// TIA Portal V19 program export: 4 tag tables, 24 data types, 99 data blocks, 53 code blocks (in call order from the OBs), 0 instance data blocks

VAR_GLOBAL   // PLC tag table "Default tag table"
   Tag_111 AT %MW1 : Int;
   di_1 AT %I0.0 : Bool;
   di_2 AT %I0.1 : Bool;
   ai_raw_01 AT %IW272 : Int;
   ai_raw_02 AT %IW274 : Int;
   ai_raw_03 AT %IW276 : Int;
   ai_raw_04 AT %IW278 : Int;
END_VAR
VAR_GLOBAL CONSTANT   // user constants
   C_HW_MAX : Int := 27648;
   C_HW_MIN : Int := 0;
   C_DIAG_OVER : Real := 1.1759;
   C_DIAG_UNDER : Real := -0.1759;
END_VAR

VAR_GLOBAL   // PLC tag table "Tag table_1"
   r1 AT %M20.0 : Bool;
   tr1 AT %M20.1 : Bool;
   r2 AT %M20.2 : Bool;
   tr2 AT %M20.3 : Bool;
   r3 AT %M20.4 : Bool;
   tr3 AT %M20.5 : Bool;
   r4 AT %M20.6 : Bool;
   tr4 AT %M20.7 : Bool;
   r5 AT %M21.0 : Bool;
   tr5 AT %M21.1 : Bool;
   r6 AT %M21.2 : Bool;
   tr6 AT %M21.3 : Bool;
   r7 AT %M21.4 : Bool;
   tr7 AT %M21.5 : Bool;
   r8 AT %M21.6 : Bool;
   tr8 AT %M21.7 : Bool;
   r9 AT %M22.0 : Bool;
   tr9 AT %M22.1 : Bool;
   r10 AT %M22.2 : Bool;
   tr10 AT %M22.3 : Bool;
   r11 AT %M22.4 : Bool;
   tr11 AT %M22.5 : Bool;
   r12 AT %M22.6 : Bool;
   tr12 AT %M22.7 : Bool;
   r13 AT %M23.0 : Bool;
   tr13 AT %M23.1 : Bool;
   r14 AT %M23.2 : Bool;
   tr14 AT %M23.3 : Bool;
   r15 AT %M23.4 : Bool;
   tr15 AT %M23.5 : Bool;
END_VAR

VAR_GLOBAL   // PLC tag table "Tag table_2"
   Pol_sklad_sens AT %IW40 : Int;
   Pol_sens AT %IW42 : Int;
END_VAR

VAR_GLOBAL   // PLC tag table "Tag tanks"
END_VAR
VAR_GLOBAL CONSTANT   // user constants
   c_Count_TRN : Int := 3;
   c_Count_POL : Int := 10;
   c_Count_BUL : Int := 4;
   c_Count_MOL : Int := 12;
END_VAR

TYPE "UDT_AI_Alarm_Conf"
VERSION : 0.1
   STRUCT
      En_Alarm : Struct
         HiHi { S7_SetPoint := 'True'} : Bool;
         Hi { S7_SetPoint := 'True'} : Bool;
         Lo { S7_SetPoint := 'True'} : Bool;
         LoLo { S7_SetPoint := 'True'} : Bool;
         Latch_Enable { S7_SetPoint := 'True'} : Bool;   // 1 = Включена фиксация аварий (до нажатия Reset)
         Pad_Bit_5 { S7_SetPoint := 'True'} : Bool;   // Резерв
         Pad_Bit_6 { S7_SetPoint := 'True'} : Bool;   // Резерв
         Pad_Bit_7 { S7_SetPoint := 'True'} : Bool;   // Резерв
      END_STRUCT;
      HiHi { S7_SetPoint := 'True'} : Real;
      Hi { S7_SetPoint := 'True'} : Real;
      Lo { S7_SetPoint := 'True'} : Real;
      LoLo { S7_SetPoint := 'True'} : Real;
      Delay_HiHi { S7_SetPoint := 'True'} : Int;
      Delay_Hi { S7_SetPoint := 'True'} : Int;
      Delay_Lo { S7_SetPoint := 'True'} : Int;
      Delay_LoLo { S7_SetPoint := 'True'} : Int;
      Hysteresis { S7_SetPoint := 'True'} : Real;
   END_STRUCT;

END_TYPE

TYPE "UDT_AI_Conf"
VERSION : 0.1
   STRUCT
      Mode { S7_SetPoint := 'True'} : Word := 16#0010;   // ПО УМОЛЧАНИЮ: Взведен Bit 4 (Final Clamp)
      Scale_Min { S7_SetPoint := 'True'} : Real := 0.0;   // Мин. физической шкалы
      Scale_Max { S7_SetPoint := 'True'} : Real := 100.0;   // Макс. физической шкалы
      Calib_mA_Min { S7_SetPoint := 'True'} : Real := 4.0;   // Ток при Scale_Min
      Calib_mA_Max { S7_SetPoint := 'True'} : Real := 20.0;   // Ток при Scale_Max
      Cutoff { S7_SetPoint := 'True'} : Real := 0.02;   // Порог отсечения шума около нуля
      FilterTime_ms { S7_SetPoint := 'True'} : Int := 2000;   // Время фильтра PT1 в миллисекундах (0..32000) --- Границы железа ---
      HW_Min { S7_SetPoint := 'True'} : Int := "C_HW_MIN";   // Аппаратный минимум
      HW_Max { S7_SetPoint := 'True'} : Int := "C_HW_MAX";   // Аппаратный максимум
   END_STRUCT;

END_TYPE

TYPE "UDT_AI_Config"
VERSION : 0.1
   STRUCT
      Mode : Word := 16#0010;   // ПО УМОЛЧАНИЮ: Взведен Bit 4 (Final Clamp)
      Scale_Min : Real := 0.0;   // Мин. физической шкалы
      Scale_Max : Real := 100.0;   // Макс. физической шкалы
      Calib_mA_Min : Real := 4.0;   // Ток при Scale_Min
      Calib_mA_Max : Real := 20.0;   // Ток при Scale_Max
      Cutoff : Real := 0.02;   // Порог отсечения шума около нуля
      FilterTime_ms : Int := 2000;   // Время фильтра PT1 в миллисекундах (0..32000) --- Границы железа ---
      HW_Min : Int := "C_HW_MIN";   // Аппаратный минимум
      HW_Max : Int := "C_HW_MAX";   // Аппаратный максимум
   END_STRUCT;

END_TYPE

TYPE "UDT_AI_Out"
VERSION : 0.1
   STRUCT
      Raw : Int;   // Сырой код с модуля (PIW)
      Value_mA : Real;   // Расчетный ток (мА)
      Value_Unclamped : Real;   // Чистая физика (ДО клампа и ДО фильтра)
      Value_Scaled : Real;   // Физика ПОСЛЕ клампа (ограниченная шкалой)
      Value_Filtered : Real;   // Финальное сглаженное значение (для HMI и алармов)
      Status : Struct
         WireBreak : Bool;
         Underrange : Bool;
         Overrange : Bool;
         Overflow : Bool;
         Sim_Active : Bool;
         ConfigError : Bool;
         Pad_Bit_6 : Bool;   // Выравнивание
         Pad_Bit_7 : Bool;   // Выравнивание
         Pad_Byte : Byte;   // Выравнивание структуры до 1 Word
      END_STRUCT;
   END_STRUCT;

END_TYPE

TYPE "UDT_AI_Status"
VERSION : 0.1
// -----------------------------------------------------------------------------
// 2. АВТОНОМНЫЙ СТАТУС (2 БАЙТА / 1 WORD)
// -----------------------------------------------------------------------------
   STRUCT
      WireBreak : Bool;   // +0.0 | Wire break (< -4864)
      Underrange : Bool;   // +0.1 | Signal < 0 mA, but alive
      Overrange : Bool;   // +0.2 | Signal > 20 mA
      Overflow : Bool;   // +0.3 | Short circuit (> 22.8 mA)
      Sim_Active : Bool;   // +0.4 | Simulation mode ON
      ConfigError : Bool;   // +0.5 | Bad settings in UDT_Config
      Pad_Bit_6 : Bool;   // +0.6
      Pad_Bit_7 : Bool;   // +0.7
      Pad_Byte : Byte;   // +1.0 | Alignment for S7-300
   END_STRUCT;

END_TYPE

TYPE "UDT_Alarm_Config"
VERSION : 1.0
   STRUCT
      En_Alarm : Struct
         HiHi         : Bool;
         Hi           : Bool;
         Lo           : Bool;
         LoLo         : Bool;
         Latch_Enable : Bool;  // 1 = Включена фиксация аварий (до нажатия Reset)
         Pad_Bit_5    : Bool;  // Резерв
         Pad_Bit_6    : Bool;  // Резерв
         Pad_Bit_7    : Bool;  // Резерв
      END_STRUCT;
      HiHi       : Real;
      Hi         : Real;
      Lo         : Real;
      LoLo       : Real;
      Delay_HiHi : Int;
      Delay_Hi   : Int;
      Delay_Lo   : Int;
      Delay_LoLo : Int;
      Hysteresis : Real;
   END_STRUCT;
END_TYPE

TYPE "UDT_Alarm_Out"
VERSION : 2.0
   STRUCT
      // --- Байт 0 (Аварии) ---
      HiHi         : Bool;
      Hi           : Bool;
      Lo           : Bool;
      LoLo         : Bool;
      Pad_Bit_4    : Bool; // Резерв
      Pad_Bit_5    : Bool; // Резерв
      Pad_Bit_6    : Bool; // Резерв
      Pad_Bit_7    : Bool; // Резерв
      
      // --- Байт 1 (Статусы для HMI) ---
      En_HiHi         : Bool;
      En_Hi           : Bool;
      En_Lo           : Bool;
      En_LoLo         : Bool;
      En_Latch_Enable : Bool; // Статус фиксации
      En_Pad_Bit_5    : Bool; // Резерв
      En_Pad_Bit_6    : Bool; // Резерв
      En_Pad_Bit_7    : Bool; // Резерв
   END_STRUCT;
END_TYPE

TYPE "UDT_DI_Alarm_Conf"
VERSION : 0.1
// =============================================================================
// СТРУКТУРЫ ДЛЯ ДИСКРЕТНОГО АЛАРМА (FB_DI_Alarm)
// =============================================================================
   STRUCT
      En_Alarm : Bool;   // 1 = Разрешение контроля аварии
      Invert : Bool;   // 0 = NO (TRUE = Авария), 1 = NC (FALSE = Авария)
      Latch_Enable : Bool;   // 1 = Фиксация аварии (требует сброса кнопкой Reset)
      Pad_Bit_3 : Bool;   // Резерв
      Pad_Bit_4 : Bool;   // Резерв
      Pad_Bit_5 : Bool;   // Резерв
      Pad_Bit_6 : Bool;   // Резерв
      Pad_Bit_7 : Bool;   // Резерв
      Pad_Byte : Byte;   // Выравнивание
      Delay : Int;   // Задержка срабатывания (в СЕКУНДАХ)
   END_STRUCT;

END_TYPE

TYPE "UDT_DI_Conf"
VERSION : 0.1
   STRUCT
      Mode { S7_SetPoint := 'True'} : Int;   // Режим: 0=Прямой, 1=С фильтром (Прямой), 2=С фильтром (Инверсный)
      FilterTime { S7_SetPoint := 'True'} : Int;   // Время антидребезга (мс), макс. 32767 мс
   END_STRUCT;

END_TYPE

TYPE "UDT_DI_Out"
VERSION : 0.1
// =============================================================================
// СТРУКТУРЫ ДЛЯ ОБРАБОТКИ ДИСКРЕТНОГО ВХОДА (FB_DI)
// =============================================================================
   STRUCT
      Value : Bool;   // Обработанное состояние входа (после антидребезга)
      Pad_Bit_1 : Bool;   // Резерв
      Pad_Bit_2 : Bool;   // Резерв
      Pad_Bit_3 : Bool;   // Резерв
      Pad_Bit_4 : Bool;   // Резерв
      Pad_Bit_5 : Bool;   // Резерв
      Pad_Bit_6 : Bool;   // Резерв
      Pad_Bit_7 : Bool;   // Резерв
      Pad_Byte : Byte;   // Выравнивание до слова (Word) для SCADA
   END_STRUCT;

END_TYPE

TYPE "UDT_HMI_SmallTank"
TITLE = Данные малого танка для HMI
VERSION : 0.1
//Описание:
//        Плоская структура малого танка для обмена с панелью оператора.
//        Статусные слова развернуты побитово с жестким выравниванием 
//        до 16 бит (WORD) для прямого маппинга в библиотеку WinCC.
   STRUCT
      Level_m : Real;   // Текущий уровень
      Volume_m3 : Real;   // Рассчитанный объем
      Weight_t : Real;   // Рассчитанная масса в тоннах
      Percent_prc : Real;   // Уровень в процентах --- Развернутое слово Status_Alarms (Ровно 2 байта) ---
      Status_Alarms : Struct
         DI : Bool;   // ПЛК Бит 0.0 -> WinCC Бит 8
         HH : Bool;   // ПЛК Бит 0.1 -> WinCC Бит 9
         H : Bool;   // ПЛК Бит 0.2 -> WinCC Бит 10
         L : Bool;   // ПЛК Бит 0.3 -> WinCC Бит 11
         LL : Bool;   // ПЛК Бит 0.4 -> WinCC Бит 12
         Pad_0_5 : Bool;   // Выравнивание
         Pad_0_6 : Bool;   // Выравнивание
         Pad_0_7 : Bool;   // Выравнивание
         Pad_Byte : Byte;   // Резервный младший байт (WinCC Биты 0..7) --- Развернутое слово Status_AI (Ровно 2 байта) ---
      END_STRUCT;
      Status_AI : Struct
         WireBreak : Bool;   // ПЛК Бит 0.0 -> WinCC Бит 8
         Underrange : Bool;   // ПЛК Бит 0.1 -> WinCC Бит 9
         Overrange : Bool;   // ПЛК Бит 0.2 -> WinCC Бит 10
         Overflow : Bool;   // ПЛК Бит 0.3 -> WinCC Бит 11
         ConfigError : Bool;   // ПЛК Бит 0.4 -> WinCC Бит 12
         Pad_0_5 : Bool;   // Выравнивание
         Pad_0_6 : Bool;   // Выравнивание
         Pad_0_7 : Bool;   // Выравнивание
         Pad_Byte : Byte;   // Резервный младший байт (WinCC Биты 0..7) --- Развернутое слово Cmd_Word (Ровно 2 байта) ---
      END_STRUCT;
      Cmd : Struct
         Reset : Bool;   // ПЛК Бит 0.0 -> WinCC Бит 8 (Кнопка сброса)
         Pad_0_1 : Bool;   // Выравнивание
         Pad_0_2 : Bool;   // Выравнивание
         Pad_0_3 : Bool;   // Выравнивание
         Pad_0_4 : Bool;   // Выравнивание
         Pad_0_5 : Bool;   // Выравнивание
         Pad_0_6 : Bool;   // Выравнивание
         Pad_0_7 : Bool;   // Выравнивание
         Pad_Byte : Byte;   // Резервный младший байт (WinCC Биты 0..7)
      END_STRUCT;
      Spare_Real_1 : Real;   // Резерв для сохранения смещений
   END_STRUCT;

END_TYPE

TYPE "UDT_HMI_Whouse"
TITLE = Сводка склада для HMI
{ S7_Optimized_Access := 'FALSE' }
AUTHOR : S7A_Lib
FAMILY : HMI_Type
VERSION : 0.1
// ==============================================================================
// Описание: Агрегированные данные склада (тоталы, счетчики, глобальные 
//           статусы) для отображения на главном экране WinCC.
// ==============================================================================
    STRUCT
        Total_Volume_m3 : REAL;   // Суммарный объем продукта на складе
        Total_Weight_t : REAL;    // Суммарная масса (тонны)
        Total_Ullage_m3 : REAL;   // Доступное свободное место (м3)
        Tanks_In_Alarm : INT;     // Количество танков в состоянии аварии
        
        // --- Глобальные статусы склада (Ровно 2 байта) ---
        Status_Word : STRUCT 
            Comm_Error : BOOL;    // ПЛК Бит 0.0 -> WinCC Бит 8 (Ошибка связи с периферией)
            Global_Alarm : BOOL;  // ПЛК Бит 0.1 -> WinCC Бит 9 (Есть активные аварии)
            Pad_0_2 : BOOL;       // Выравнивание
            Pad_0_3 : BOOL;       // Выравнивание
            Pad_0_4 : BOOL;       // Выравнивание
            Pad_0_5 : BOOL;       // Выравнивание
            Pad_0_6 : BOOL;       // Выравнивание
            Pad_0_7 : BOOL;       // Выравнивание
            Pad_Byte : BYTE;      // Резервный младший байт (WinCC Биты 0..7)
        END_STRUCT;
        
        // --- Глобальные команды склада (Ровно 2 байта) ---
        Cmd_Word : STRUCT
            Reset_All : BOOL;     // ПЛК Бит 0.0 -> WinCC Бит 8 (Глобальный сброс аварий)
            Pad_0_1 : BOOL;       // Выравнивание
            Pad_0_2 : BOOL;       // Выравнивание
            Pad_0_3 : BOOL;       // Выравнивание
            Pad_0_4 : BOOL;       // Выравнивание
            Pad_0_5 : BOOL;       // Выравнивание
            Pad_0_6 : BOOL;       // Выравнивание
            Pad_0_7 : BOOL;       // Выравнивание
            Pad_Byte : BYTE;      // Резервный младший байт (WinCC Биты 0..7)
        END_STRUCT;
        
        Spare_Real_1 : REAL;      // Резерв для сохранения смещений
    END_STRUCT;
END_TYPE

TYPE "UDT_SIWA_CS"
VERSION : 0.0
   STRUCT
      i_DB_Lenght : Int := 222;
      i_MaxLifeBitCyc : Int := 500;
      i_SFC_ERR_C : Word;
      i_CMD_INPUT : Int;
      bo_CMD_TRIGGER : Bool;
      bo_CMD_IN_PROGRESS : Bool;
      bo_CMD_FINISHED_OK : Bool;
      bo_CMD_ERR : Bool;
      b_CMD_ERR_CODE : Byte;
      i_PRESET_TARE : Int;
      b_SELECT_PROC_VAL : Byte;
      b_SELECTED_PROC_VAL : Byte;
      i_PROCESS_VALUE : Int;
      b_INFO_REFRESH_COUNT : Byte;
      w_SCALE_STATUS : Word;
      b_OPR_ERR_MSG : Byte;
      bo_FB_ERR : Bool;
      b_FB_ERR_CODE : Byte;
      bo_START_UP_IN_PROGRESS : Bool;
      s_CMD1 : Struct
         i_CMD1_Code : Int;
         bo_CMD1_Trigger : Bool;
         bo_CMD1_InProgress : Bool;
         bo_CMD1_FinishedOk : Bool;
         bo_CMD1_FinishedError : Bool;
      END_STRUCT;
      s_CMD2 : Struct
         i_CMD2_Code : Int;
         bo_CMD2_Trigger : Bool;
         bo_CMD2_InProgress : Bool;
         bo_CMD2_FinishedOk : Bool;
         bo_CMD2_FinishedError : Bool;
      END_STRUCT;
      s_CMD3 : Struct
         i_CMD3_Code : Int;
         bo_CMD3_Trigger : Bool;
         bo_CMD3_InProgress : Bool;
         bo_CMD3_FinishedOk : Bool;
         bo_CMD3_FinishedError : Bool;
      END_STRUCT;
      w_DB_RES92 : Word;
      w_DB_RES93 : Word;
      w_DB_RES94 : Word;
      w_DB_RES95 : Word;
      w_DB_RES96 : Word;
      w_DB_RES97 : Word;
      w_INT_USE : Word;
      s_JUST_DAT : Struct
         w_CALIB_DIGITS0 : Word;
         w_CALIB_DIGITS1 : Word := W#16#EA60;
         w_CALIB_DIGITS2 : Word;
         i_CALIB_WEIGHT1 : Int := 2000;
         i_CALIB_WEIGHT2 : Int;
         b_SIGNAL_RANGE : Byte := B#16#2;
         b_FILT_TYPE : Byte;
         b_FILT_FREQ : Byte := B#16#4;
         b_FILT_DEPTH : Byte := B#16#F;
         s_SCALE_ID : String[10] := 'SIWAREX XX';
         i_MIN_WR : Int := 20;
         i_MAX_WR : Int := 2000;
         i_INCREMENT_WR : Int := 1;
         i_WEIGHT_ST_STILL : Int := 10;
         t_TIME_ST_STILL1 : Time := T#1S;
         b_DEC_POINT : Byte := B#16#2;
         b_ZERO_NEG_VALUE : Byte := B#16#1;
         b_ZERO_POS_VALUE : Byte := B#16#3;
         b_TARA_MAX : Byte := B#16#64;
         i_Reserve : Int;
         s_LEGAL_TRADE : String[4] := '----';
         s_WEGHT_UNIT : String[4] := 'kg  ';
      END_STRUCT;
      s_LIMIT_PARA : Struct
         i_LIMIT1_ON : Int := 400;
         i_LIMIT1_OFF : Int := 220;
         i_LIMIT2_ON : Int := 1000;
         i_LIMIT2_OFF : Int := 980;
         bo_LIMIT1_PARA : Bool;
         bo_LIMIT2_PARA : Bool;
         b_Reserve : Byte;
      END_STRUCT;
      s_MODUL_INFO_DATA : Struct
         s_MODUL_NAME : String[10];
         s_ORDER_NUM : String[20];
         w_VERSION_HW : Word;
         s_VERSION_FW : String[4];
         w_CRC_CHECK : Word;
      END_STRUCT;
      s_TARE_CONTROL : Struct
         i_TARE_VALUE : Int;
      END_STRUCT;
      s_INTERNAL_PROC_VAL : Struct
         w_CRC_CHECK : Word;
         b_Reserve : Byte;
         bo_PRESET_TARA : Bool;
         d_TARA_X_100 : DInt;
         d_ZERO_X_100 : DInt;
      END_STRUCT;
      s_PROCESS_VALUES : Struct
         w_CRC_CHECK : Word;
         bo_STA_WRI_PROT : Bool;
         bo_STA_WR_MIN : Bool;
         bo_STA_Reserve1 : Bool;
         bo_STA_Reserve2 : Bool;
         bo_STA_Reserve3 : Bool;
         bo_STA_Reserve4 : Bool;
         bo_STA_Reserve5 : Bool;
         bo_STA_ERROR_ON : Bool;
         bo_STA_LIMIT1_ON : Bool;
         bo_STA_LIMIT2_ON : Bool;
         bo_STA_TARED : Bool;
         bo_STA_TARED_BY_MANUAL : Bool;
         bo_STA_MAX_9E : Bool;
         bo_STA_025_D_ZERO : Bool;
         bo_STA_ST_STAND_SCALE_ON : Bool;
         bo_STA_SCALE_CALIBRATED : Bool;
         b_OPR_ERR_MSG : Byte;
         b_Reserve : Byte;
         i_GROSS_WEIGHT_PROC : Int;
         i_NET_WEIGHT_PROC : Int;
         i_TARE_WEIGHT_PROC : Int;
         i_GROSS_NET_VALUE : Int;
         d_GROSS_NET_VALUE_10X : DInt;
         i_TARE_VALUE : Int;
         i_ADC_DIGIT : Int;
         i_ADC_DIGIT_FILTER : Int;
         s_WEIGHT_ASCII : String[14];
         i_MILISEC : Int;
         b_SECONDS : Byte;
         b_MINUTE : Byte;
         i_HOURS : Int;
      END_STRUCT;
      i_DB_Lenght1 : Int := 222;
   END_STRUCT;

END_TYPE

TYPE "UDT_Siwarex_Core"
TITLE = Данные весового модуля Siwarex
VERSION : 0.2
//Описание:
//        Базовая структура для работы с весовыми модулями Siwarex.
//        Разделены операционные ошибки (модуля) и ошибки драйвера (FB).
    STRUCT
        Weight_Gross_kg : REAL;    // Брутто (полный вес)
        Weight_Net_kg : REAL;      // Нетто (чистый вес продукта)
        Weight_Tare_kg : REAL;     // Тара (вес пустой емкости)
        
        // --- Диагностика: Аппаратная ошибка модуля (из b_OPR_ERR_MSG) ---
        // 17 - Выход за максимальный предел взвешивания.
        // 19 - Перегруз АЦП (ADC overrange).
        // 20 - Недогруз АЦП (сигнал ушел далеко в минус).
        // 22 - Ошибка команды: весы не стабильны (жидкость плещется).
        // 31 - Обрыв провода тензодатчика (Wire break).
        Error_Op_Msg : INT;        
        
        // --- Диагностика: Ошибка драйвера ПЛК (из b_FB_ERR_CODE) ---
        // 1 - Watchdog тайм-аут (нет ответа от модуля на запрос данных).
        // 2 - Ошибка системной функции (SFC) RD_REC или WR_REC.
        // 3 - Некорректный номер команды в буфере или неверная длина DB.
        Error_FB_Code : INT;       
        
        // --- Статусы весов (Ровно 2 байта) ---
        Status : STRUCT
            Standstill : BOOL;     // ПЛК Бит 0.0 -> WinCC Бит 8 (Весы в покое)
            Limit_1 : BOOL;        // ПЛК Бит 0.1 -> WinCC Бит 9 (Предел 1)
            Limit_2 : BOOL;        // ПЛК Бит 0.2 -> WinCC Бит 10 (Предел 2)
            Fault_HW : BOOL;       // ПЛК Бит 0.3 -> WinCC Бит 11 (Аппаратная ошибка)
            Limit_Max : BOOL;      // ПЛК Бит 0.4 -> WinCC Бит 12 (Перегруз)
            Comm_Fault : BOOL;     // ПЛК Бит 0.5 -> WinCC Бит 13 (Watchdog: потеря связи)
            Fault_FB : BOOL;       // ПЛК Бит 0.6 -> WinCC Бит 14 (Ошибка драйвера)
            Pad_0_7 : BOOL;        // Выравнивание
            Pad_Byte : BYTE;       // Резервный младший байт (WinCC Биты 0..7)
        END_STRUCT;
        
        // --- Команды с HMI (Ровно 2 байта) ---
        Cmd : STRUCT
            Zero : BOOL;           // ПЛК Бит 0.0 -> WinCC Бит 8 (Установка нуля)
            Tare : BOOL;           // ПЛК Бит 0.1 -> WinCC Бит 9 (Тарирование)
            ResetError : BOOL;     // ПЛК Бит 0.2 -> WinCC Бит 10 (Сброс ошибки)
            Pad_0_3 : BOOL;        // Выравнивание
            Pad_0_4 : BOOL;        // Выравнивание
            Pad_0_5 : BOOL;        // Выравнивание
            Pad_0_6 : BOOL;        // Выравнивание
            Pad_0_7 : BOOL;        // Выравнивание
            Pad_Byte : BYTE;       // Резервный младший байт (WinCC Биты 0..7)
        END_STRUCT;
        
        Spare_Real_1 : REAL;       // Резерв
    END_STRUCT;
END_TYPE

TYPE "UDT_Sys_Info"
VERSION : 0.1
// ===============================================================
// Master Project: S7C_Master_AI_Test (S7-300 COMPLIANT)
// Platform: S7-300 / IM 151-8
// FIX: No FBs in Temp/Global DB. Using Multi-instance in Wrapper FB.
// Encoding: UTF-8 with BOM
// ===============================================================
// 1. DATA TYPES (UDTs)
   STRUCT
      FirstScan { ExternalVisible := 'False'} : Bool;
      CycleTime_ms_INT { ExternalVisible := 'False'} : Int;
      CycleTime_ms_REAL { ExternalVisible := 'False'} : Real;
   END_STRUCT;

END_TYPE

TYPE "UDT_Tank_Calc"
VERSION : 0.1
// Технологические показатели (результаты расчетов)
   STRUCT
      Weight_t : Real;   // Текущий вес (тонны)
      Volume_m3 : Real;   // Текущий объем (м3)
      Ullage_m3 : Real;   // Свободное место (м3)
      Level_Pct : Real;   // Уровень (0.0 - 100.0 %)
      Level_m : Real;   // Уровень (мм)
   END_STRUCT;

END_TYPE

TYPE "UDT_Tank_Full"
VERSION : 0.1
// Полная структура одного танка (Агрегатор)
   STRUCT
      AI_Conf : "UDT_AI_Conf";   // Настройки входа (Mode, Sim и т.д.)
      AI_Out : "UDT_AI_Out";   // Результаты фильтрации (Value_Filtered)
      AI_Alarm_Conf : "UDT_AI_Alarm_Conf";   // Уставки (HH, H, L, LL)
      AI_Alarm : "UDT_AI_Alarm";   // Статус аварий по AI --- Секция DI (твои структуры) ---
      DI_Conf : "UDT_DI_Conf";   // Настройки фильтра дребезга
      DI_Out : "UDT_DI_Out";   // Состояние после фильтра
      DI_Alarm_Conf : "UDT_DI_Alarm_Conf";   // Настройки аларма ВУ (Latch, Delay)
      DI_Alarm : "UDT_DI_Alarm";   // Статус аварии ВУ --- Технологическая секция ---
      Geom : "UDT_Tank_Geom";   // Паспорт танка
      Calc : "UDT_Tank_Calc";   // Сиропная математика
      Cmd : "UDT_Tank_Cmd";   // Команды
   END_STRUCT;

END_TYPE

TYPE "UDT_Tank_Geom"
VERSION : 0.1
// Физические параметры и константы емкости
   STRUCT
      Height_Full { S7_SetPoint := 'True'} : Real;   // Высота танка от 0 до 100% (мм)
      Sensor_Offset { S7_SetPoint := 'True'} : Real;   // Смещение датчика относительно дна (мм)
      Density { S7_SetPoint := 'True'} : Real;   // Плотность продукта (кг/м3)
      Max_Volume { S7_SetPoint := 'True'} : Real;   // Максимальный объем (м3)
   END_STRUCT;

END_TYPE

TYPE "UDT_AI_Alarm"
VERSION : 0.1
   STRUCT
      HiHi : Bool;
      Hi : Bool;
      Lo : Bool;
      LoLo : Bool;
      Pad_Bit_4 : Bool;   // Резерв
      Pad_Bit_5 : Bool;   // Резерв
      Pad_Bit_6 : Bool;   // Резерв
      Pad_Bit_7 : Bool;   // Резерв --- Байт 1 (Статусы для HMI) ---
      En_HiHi : Bool;
      En_Hi : Bool;
      En_Lo : Bool;
      En_LoLo : Bool;
      En_Latch_Enable : Bool;   // Статус фиксации
      En_Pad_Bit_5 : Bool;   // Резерв
      En_Pad_Bit_6 : Bool;   // Резерв
      En_Pad_Bit_7 : Bool;   // Резерв
   END_STRUCT;

END_TYPE

TYPE "UDT_Analog_In"
VERSION : 0.1
   STRUCT
      IW_HW_UpLevel : Int := 27648;
      IW_HW_LowLevel : Int := 0;
      IDW_UpLevel : Real;
      IDW_LowLevel : Real;
      IDW_HiHi : Real;
      IDW_Hi : Real;
      IDW_Lo : Real;
      IDW_Lolo : Real;
      IW_DelayON_HiHi : Int;
      IW_DelayON_Hi : Int;
      IW_DelayON_Lo : Int;
      IW_DelayON_LoLo : Int;
      IDW_Simulation_Value : Real;
      IW_Time_Filter : Int;
      IW_CTW : Array[0..15] of Bool;
      IDW_K_Mult : Real := 1.0;
      IDW_DeadZone : Real;
      IBt_Enable_ControlLevel : Array[0..7] of Bool;
      IBt_Block_ControlLevel : Array[0..7] of Bool;
      QW_STW : Array[0..15] of Bool;
      QW_HWValue : Int;
      QDW_ScalledValue : Real;
      QDW_Message : Array[0..16] of Bool;
   END_STRUCT;

END_TYPE

TYPE "UDT_DI_Alarm"
VERSION : 0.1
   STRUCT
      Alarm : Bool;   // Состояние аварии (с учетом задержки и фиксации)
      Pad_Bit_1 : Bool;   // Резерв
      Pad_Bit_2 : Bool;   // Резерв
      Pad_Bit_3 : Bool;   // Резерв
      Pad_Bit_4 : Bool;   // Резерв
      Pad_Bit_5 : Bool;   // Резерв
      Pad_Bit_6 : Bool;   // Резерв
      Pad_Bit_7 : Bool;   // Резерв --- Байт 1 (Статусы для HMI) ---
      En_Alarm : Bool;   // Статус HMI: Авария включена и не заблокирована
      Latch_Enable : Bool;   // Статус HMI: Включена фиксация
      Input_Raw : Bool;   // Диагностика HMI: Физическое состояние входа
      Input_Inv : Bool;   // Диагностика HMI: Состояние после учета инверсии
      Pad_En_4 : Bool;   // Резерв
      Pad_En_5 : Bool;   // Резерв
      Pad_En_6 : Bool;   // Резерв
      Pad_En_7 : Bool;   // Резерв
   END_STRUCT;

END_TYPE

TYPE "UDT_Log_Record"
VERSION : 0.1
   STRUCT
      Timestamp : Date_And_Time; // 8 байт
      Whouse_ID : Byte;          // ID склада (1..4)
      Tank_Index : Byte;         // Номер танка в массиве
      Level_m : Real;            // Уровень из Calc.Level_m
      Weight_t : Real;           // Вес из Calc.Weight_t
      Status_Bits : Byte;        // Упакованные аварии (HiHi, Hi, Lo, LoLo)
      Pad_Byte : Byte;           // Выравнивание до четного числа байт
   END_STRUCT;
END_TYPE

TYPE "UDT_SIWA_Cmd"
VERSION : 0.1
   STRUCT
      i_Code : Int;
      bo_Trigger : Bool;
      bo_InProgress : Bool;
      bo_FinishedOk : Bool;
      bo_FinishedError : Bool;
   END_STRUCT;

END_TYPE

TYPE "UDT_Tank_Cmd"
VERSION : 0.1
// Команды управления танком
   STRUCT
      ResetError : Bool;   // Сброс зафиксированных аварий (Latch)
      CalibrateDensity : Bool;   // Запрос на автокалибровку плотности (резерв)
      Spare_02 : Bool;
      Spare_03 : Bool;
      Spare_04 : Bool;
      Spare_05 : Bool;
      Spare_06 : Bool;
      Spare_07 : Bool;
   END_STRUCT;

END_TYPE

DATA_BLOCK "DB_Global"
{ S7_Optimized_Access := 'FALSE' }
VERSION : 0.1
// 2. GLOBAL DATA (Pure Data only)
   STRUCT 
      Sys : "UDT_Sys_Info";
   END_STRUCT;


BEGIN

END_DATA_BLOCK

DATA_BLOCK "DB_IO_MAP"
{ S7_Optimized_Access := 'FALSE' }
VERSION : 0.1
   STRUCT 
      AI_TRN_Tank_1 : Int;
      AI_TRN_WTank_2 : Int;
      AI_TRN_WTank_3 : Int;
      DI_TRN_Tank_1 : Bool;
      DI_TRN_WTank_2 : Bool;
      DI_TRN_WTank_3 : Bool;
      AI_POL_Tank_1 : Int;
      AI_POL_Tank_2 : Int;
      AI_POL_Tank_3 : Int;
      DI_POL_Tank_1 : Bool;
      DI_POL_Tank_2 : Bool;
      DI_POL_Tank_3 : Bool;
   END_STRUCT;


BEGIN

END_DATA_BLOCK

DATA_BLOCK "DB_Logic_IDB"
{ S7_Optimized_Access := 'FALSE' }
VERSION : 0.1
// 7. MAIN CALL
"FB_Station_Logic"

BEGIN

END_DATA_BLOCK

DATA_BLOCK "DB_Test_IO"
{ S7_Optimized_Access := 'FALSE' }
VERSION : 0.1
   STRUCT 
      Sim_Enable_Saw : Bool;
      Sim_Enable_Noise : Bool;
      Sim_Saw_Speed : Real;
      Sim_Noise_Amp : Int;
      Sim_Noise_Hz : Real;
      Raw_Final : Int;
      Reset_Alarms : Bool;
      Config : Array[1..2] of "UDT_AI_Config";
      Out : Array[1..2] of "UDT_AI_Out";
      Alarm_Cfg : Array[1..2] of "UDT_Alarm_Config";
      Alarm_Out : Array[1..2] of "UDT_Alarm_Out";
      Raw_Start { S7_SetPoint := 'True'} : Int;
      Raw_Min : Int;
      Raw_Max : Int;
   END_STRUCT;


BEGIN
   Sim_Saw_Speed := 500.0;
   Sim_Noise_Amp := 200;
   Sim_Noise_Hz := 2.0;
   Config[1].Scale_Max := 100.0;
   Alarm_Cfg[1].HiHi := 90.0;
   Alarm_Cfg[1].Delay_HiHi := 2;
   Raw_Min := 0;
   Raw_Max := 27222;

END_DATA_BLOCK

DATA_BLOCK "iDB_BUL_Tank_Log_2"
{ S7_Optimized_Access := 'FALSE' }
AUTHOR : Gemini
FAMILY : Archive
VERSION : 1.2
NON_RETAIN
"FB_Tank_Logic"

BEGIN

END_DATA_BLOCK

DATA_BLOCK "iDB_MOL_Tank_Log_1"
{ S7_Optimized_Access := 'FALSE' }
AUTHOR : Gemini
FAMILY : Archive
VERSION : 1.2
NON_RETAIN
"FB_Tank_Logic"

BEGIN

END_DATA_BLOCK

DATA_BLOCK "iDB_MOL_Tank_Log_10"
{ S7_Optimized_Access := 'FALSE' }
AUTHOR : Gemini
FAMILY : Archive
VERSION : 1.2
NON_RETAIN
"FB_Tank_Logic"

BEGIN

END_DATA_BLOCK

DATA_BLOCK "iDB_MOL_Tank_Log_12"
{ S7_Optimized_Access := 'FALSE' }
AUTHOR : Gemini
FAMILY : Archive
VERSION : 1.2
NON_RETAIN
"FB_Tank_Logic"

BEGIN

END_DATA_BLOCK

DATA_BLOCK "iDB_MOL_Tank_Log_2"
{ S7_Optimized_Access := 'FALSE' }
AUTHOR : Gemini
FAMILY : Archive
VERSION : 1.2
NON_RETAIN
"FB_Tank_Logic"

BEGIN

END_DATA_BLOCK

DATA_BLOCK "iDB_MOL_Tank_Log_3"
{ S7_Optimized_Access := 'FALSE' }
AUTHOR : Gemini
FAMILY : Archive
VERSION : 1.2
NON_RETAIN
"FB_Tank_Logic"

BEGIN

END_DATA_BLOCK

DATA_BLOCK "iDB_MOL_Tank_Log_4"
{ S7_Optimized_Access := 'FALSE' }
AUTHOR : Gemini
FAMILY : Archive
VERSION : 1.2
NON_RETAIN
"FB_Tank_Logic"

BEGIN

END_DATA_BLOCK

DATA_BLOCK "iDB_MOL_Tank_Log_6"
{ S7_Optimized_Access := 'FALSE' }
AUTHOR : Gemini
FAMILY : Archive
VERSION : 1.2
NON_RETAIN
"FB_Tank_Logic"

BEGIN

END_DATA_BLOCK

DATA_BLOCK "iDB_POL_Tank_Log_2"
{ S7_Optimized_Access := 'FALSE' }
AUTHOR : Gemini
FAMILY : Archive
VERSION : 1.2
"FB_Tank_Logic"

BEGIN

END_DATA_BLOCK

DATA_BLOCK "iDB_POL_Tank_Log_7"
{ S7_Optimized_Access := 'FALSE' }
AUTHOR : Gemini
FAMILY : Archive
VERSION : 1.2
NON_RETAIN
"FB_Tank_Logic"

BEGIN

END_DATA_BLOCK

DATA_BLOCK "iDB_POL_Tank_Log_9"
{ S7_Optimized_Access := 'FALSE' }
AUTHOR : Gemini
FAMILY : Archive
VERSION : 1.2
NON_RETAIN
"FB_Tank_Logic"

BEGIN

END_DATA_BLOCK

DATA_BLOCK "iDB_TRN_Tank_Log_3"
{ S7_Optimized_Access := 'FALSE' }
FAMILY : Archive
VERSION : 1.2
NON_RETAIN
"FB_Tank_Logic"

BEGIN

END_DATA_BLOCK

DATA_BLOCK "DB_Scale_CS_1"
{ S7_Optimized_Access := 'FALSE' }
VERSION : 0.1
"UDT_SIWA_CS"

BEGIN

END_DATA_BLOCK

DATA_BLOCK "DB_Scale_CS_2"
{ S7_Optimized_Access := 'FALSE' }
VERSION : 0.1
"UDT_SIWA_CS"

BEGIN

END_DATA_BLOCK

DATA_BLOCK "iDB_Map_Siwarex_Core_2"
{ S7_Optimized_Access := 'FALSE' }
AUTHOR : S7C_Lib
FAMILY : Analog
VERSION : 1.4
"FB_Map_Siwarex_Core"

BEGIN

END_DATA_BLOCK

DATA_BLOCK "DBl_SCALE_CS_1"
{ S7_Optimized_Access := 'FALSE' }
VERSION : 0.1
   STRUCT 
      Data { S7_SetPoint := 'False'} : "UDT_SIWA_CS";
   END_STRUCT;


BEGIN

END_DATA_BLOCK

DATA_BLOCK "DBl_SCALE_CS_2"
{ S7_Optimized_Access := 'FALSE' }
VERSION : 0.1
   STRUCT 
      Data { S7_SetPoint := 'False'} : "UDT_SIWA_CS";
   END_STRUCT;


BEGIN

END_DATA_BLOCK

DATA_BLOCK "DB_DateTime"
{ S7_Optimized_Access := 'FALSE' }
VERSION : 0.1
NON_RETAIN
   STRUCT 
      TimeOfDay_PLC : Time_Of_Day;
      Date_PLC : Date;
      DateTime_PLC : Date_And_Time;
      stReadDataTime_PLC : Int;
   END_STRUCT;


BEGIN
   TimeOfDay_PLC := TOD#16:14:12.371;
   Date_PLC := D#2021-11-15;
   DateTime_PLC := DT#2021-11-15-16:14:12.374;
   stReadDataTime_PLC := 0;

END_DATA_BLOCK

DATA_BLOCK "DB_Log_Buffer"
{ S7_Optimized_Access := 'FALSE' }
VERSION : 0.1
   STRUCT 
      Write_Index : Int;   // Указатель для ПЛК (куда пишем следующую запись)
      Read_Index : Int;   // Указатель для Python/1C (что считано)
      Buffer : Array[0..1999] of "UDT_Log_Record";   // Кольцевой буфер на 500 записей
   END_STRUCT;


BEGIN
   Write_Index := 0;
   Read_Index := 0;

END_DATA_BLOCK

DATA_BLOCK "DB_MAP"
{ S7_Optimized_Access := 'FALSE' }
VERSION : 0.1
NON_RETAIN
   STRUCT 
      HMI_Word_spare : DWord;
      HMI_Whouse_TRN { S7_SetPoint := 'False'} : "UDT_HMI_Whouse";
      HMI_Whouse_POL { S7_SetPoint := 'False'} : "UDT_HMI_Whouse";
      HMI_Whouse_BUL { S7_SetPoint := 'False'} : "UDT_HMI_Whouse";
      HMI_Whouse_MOL { S7_SetPoint := 'False'} : "UDT_HMI_Whouse";
      HMI_TRN_SmalTank { S7_SetPoint := 'False'} : Array[1..3] of "UDT_HMI_SmallTank";
      HMI_POL_SmalTank { S7_SetPoint := 'False'} : Array[1..10] of "UDT_HMI_SmallTank";
      HMI_BUL_SmalTank { S7_SetPoint := 'False'} : Array[1..4] of "UDT_HMI_SmallTank";
      HMI_MOL_SmalTank { S7_SetPoint := 'False'} : Array[1..12] of "UDT_HMI_SmallTank";
      Scale_CS_1 : "UDT_Siwarex_Core";
      Scale_CS_2 : "UDT_Siwarex_Core";
   END_STRUCT;


BEGIN

END_DATA_BLOCK

DATA_BLOCK "DB_Wh_BUL"
{ S7_Optimized_Access := 'FALSE' }
VERSION : 0.1
   STRUCT 
      HMI_Word_spare : DWord;
      Tank : Array[1..4] of "UDT_Tank_Full";
   END_STRUCT;


BEGIN

END_DATA_BLOCK

DATA_BLOCK "DB_Wh_MOL"
{ S7_Optimized_Access := 'FALSE' }
VERSION : 0.1
   STRUCT 
      HMI_Word_spare : DWord;
      Tank : Array[1..12] of "UDT_Tank_Full";
   END_STRUCT;


BEGIN

END_DATA_BLOCK

DATA_BLOCK "DB_Wh_POL"
{ S7_Optimized_Access := 'FALSE' }
VERSION : 0.1
   STRUCT 
      HMI_Word_spare : DWord;
      Tank : Array[1..10] of "UDT_Tank_Full";
   END_STRUCT;


BEGIN

END_DATA_BLOCK

DATA_BLOCK "DB_Wh_TRN"
{ S7_Optimized_Access := 'FALSE' }
VERSION : 0.1
   STRUCT 
      HMI_Word_spare : DWord;
      Tank : Array[1..3] of "UDT_Tank_Full";
   END_STRUCT;


BEGIN

END_DATA_BLOCK

DATA_BLOCK "Total_DB"
{ S7_Optimized_Access := 'FALSE' }
VERSION : 0.1
NON_RETAIN
   STRUCT 
      Total_Reset_HMI : Bool;
      Restart_PLC : Bool;
   END_STRUCT;


BEGIN
   Total_Reset_HMI := FALSE;
   Restart_PLC := FALSE;

END_DATA_BLOCK

DATA_BLOCK "iDB_BUL_Tank_Log_1"
{ S7_Optimized_Access := 'FALSE' }
AUTHOR : Gemini
FAMILY : Archive
VERSION : 1.2
NON_RETAIN
"FB_Tank_Logic"

BEGIN

END_DATA_BLOCK

DATA_BLOCK "iDB_BUL_Tank_Log_3"
{ S7_Optimized_Access := 'FALSE' }
AUTHOR : Gemini
FAMILY : Archive
VERSION : 1.2
NON_RETAIN
"FB_Tank_Logic"

BEGIN

END_DATA_BLOCK

DATA_BLOCK "iDB_BUL_Tank_Log_4"
{ S7_Optimized_Access := 'FALSE' }
AUTHOR : Gemini
FAMILY : Archive
VERSION : 1.2
NON_RETAIN
"FB_Tank_Logic"

BEGIN

END_DATA_BLOCK

DATA_BLOCK "iDB_MOL_Tank_Log_11"
{ S7_Optimized_Access := 'FALSE' }
AUTHOR : Gemini
FAMILY : Archive
VERSION : 1.2
NON_RETAIN
"FB_Tank_Logic"

BEGIN

END_DATA_BLOCK

DATA_BLOCK "iDB_MOL_Tank_Log_5"
{ S7_Optimized_Access := 'FALSE' }
AUTHOR : Gemini
FAMILY : Archive
VERSION : 1.2
NON_RETAIN
"FB_Tank_Logic"

BEGIN

END_DATA_BLOCK

DATA_BLOCK "iDB_MOL_Tank_Log_7"
{ S7_Optimized_Access := 'FALSE' }
AUTHOR : Gemini
FAMILY : Archive
VERSION : 1.2
NON_RETAIN
"FB_Tank_Logic"

BEGIN

END_DATA_BLOCK

DATA_BLOCK "iDB_MOL_Tank_Log_8"
{ S7_Optimized_Access := 'FALSE' }
AUTHOR : Gemini
FAMILY : Archive
VERSION : 1.2
NON_RETAIN
"FB_Tank_Logic"

BEGIN

END_DATA_BLOCK

DATA_BLOCK "iDB_MOL_Tank_Log_9"
{ S7_Optimized_Access := 'FALSE' }
AUTHOR : Gemini
FAMILY : Archive
VERSION : 1.2
NON_RETAIN
"FB_Tank_Logic"

BEGIN

END_DATA_BLOCK

DATA_BLOCK "iDB_POL_Tank_Log_1"
{ S7_Optimized_Access := 'FALSE' }
AUTHOR : Gemini
FAMILY : Archive
VERSION : 1.2
"FB_Tank_Logic"

BEGIN

END_DATA_BLOCK

DATA_BLOCK "iDB_POL_Tank_Log_10"
{ S7_Optimized_Access := 'FALSE' }
AUTHOR : Gemini
FAMILY : Archive
VERSION : 1.2
NON_RETAIN
"FB_Tank_Logic"

BEGIN

END_DATA_BLOCK

DATA_BLOCK "iDB_POL_Tank_Log_3"
{ S7_Optimized_Access := 'FALSE' }
AUTHOR : Gemini
FAMILY : Archive
VERSION : 1.2
"FB_Tank_Logic"

BEGIN

END_DATA_BLOCK

DATA_BLOCK "iDB_POL_Tank_Log_4"
{ S7_Optimized_Access := 'FALSE' }
AUTHOR : Gemini
FAMILY : Archive
VERSION : 1.2
"FB_Tank_Logic"

BEGIN

END_DATA_BLOCK

DATA_BLOCK "iDB_POL_Tank_Log_5"
{ S7_Optimized_Access := 'FALSE' }
AUTHOR : Gemini
FAMILY : Archive
VERSION : 1.2
"FB_Tank_Logic"

BEGIN

END_DATA_BLOCK

DATA_BLOCK "iDB_POL_Tank_Log_6"
{ S7_Optimized_Access := 'FALSE' }
AUTHOR : Gemini
FAMILY : Archive
VERSION : 1.2
"FB_Tank_Logic"

BEGIN

END_DATA_BLOCK

DATA_BLOCK "iDB_POL_Tank_Log_8"
{ S7_Optimized_Access := 'FALSE' }
AUTHOR : Gemini
FAMILY : Archive
VERSION : 1.2
NON_RETAIN
"FB_Tank_Logic"

BEGIN

END_DATA_BLOCK

DATA_BLOCK "iDB_TRN_Tank_Log_1"
{ S7_Optimized_Access := 'FALSE' }
AUTHOR : Gemini
FAMILY : Archive
VERSION : 1.2
NON_RETAIN
"FB_Tank_Logic"

BEGIN

END_DATA_BLOCK

DATA_BLOCK "iDB_TRN_Tank_Log_2"
{ S7_Optimized_Access := 'FALSE' }
AUTHOR : Gemini
FAMILY : Archive
VERSION : 1.2
NON_RETAIN
"FB_Tank_Logic"

BEGIN

END_DATA_BLOCK

DATA_BLOCK "iDB_Time_Trigger"
{ S7_Optimized_Access := 'FALSE' }
AUTHOR : S7A_Lib
FAMILY : Archive
VERSION : 1.1
"FB_Time_Trigger"

BEGIN

END_DATA_BLOCK

DATA_BLOCK "Pol_sklad_db"
{ S7_Optimized_Access := 'FALSE' }
VERSION : 0.1
   STRUCT 
      Pol_p : Real;
      Eror_pol_p : DWord;
      S_pol : Real;
      Weigt : Real;
      Densyty : Real;
      "1_pol" : Struct
         Weight_db : Real;
         Weight_zero : Real;
         Weight_Formula_W_T : Real;
         Visible : Bool;
         p_zero : Real;
         p_weight : Real;
         Zero_but : Bool;
         Weight_but : Bool;
         S : Real;
         Densyty : Real;
         Korect : Bool;
      END_STRUCT;
      "2_pol" : Struct
         Weight_db : Real;
         Weight_zero : Real;
         Weight_Formula_W_T : Real;
         Visible : Bool;
         p_zero : Real;
         p_weight : Real;
         Zero_but : Bool;
         Weight_but : Bool;
         S : Real;
         Densyty : Real;
         Korect : Bool;
      END_STRUCT;
      "3_pol" : Struct
         Weight_db : Real;
         Weight_zero : Real;
         Weight_Formula_W_T : Real;
         Visible : Bool;
         p_zero : Real;
         p_weight : Real;
         Zero_but : Bool;
         Weight_but : Bool;
         S : Real;
         Densyty : Real;
         Korect : Bool;
      END_STRUCT;
      "4_pol" : Struct
         Weight_db : Real;
         Weight_zero : Real;
         Weight_Formula_W_T : Real;
         Visible : Bool;
         p_zero : Real;
         p_weight : Real;
         Zero_but : Bool;
         Weight_but : Bool;
         S : Real;
         Densyty : Real;
         Korect : Bool;
      END_STRUCT;
      "5_pol" : Struct
         Weight_db : Real;
         Weight_zero : Real;
         Weight_Formula_W_T : Real;
         Visible : Bool;
         p_zero : Real;
         p_weight : Real;
         Zero_but : Bool;
         Weight_but : Bool;
         S : Real;
         Densyty : Real;
         Korect : Bool;
      END_STRUCT;
      "6_pol" : Struct
         Weight_db : Real;
         Weight_zero : Real;
         Weight_Formula_W_T : Real;
         Visible : Bool;
         p_zero : Real;
         p_weight : Real;
         Zero_but : Bool;
         Weight_but : Bool;
         S : Real;
         Densyty : Real;
         Korect : Bool;
      END_STRUCT;
      "7_pol" : Struct
         Weight_db : Real;
         Weight_zero : Real;
         Weight_Formula_W_T : Real;
         Visible : Bool;
         p_zero : Real;
         p_weight : Real;
         Zero_but : Bool;
         Weight_but : Bool;
         S : Real;
         Densyty : Real;
         Korect : Bool;
      END_STRUCT;
      "8_pol" : Struct
         Weight_db : Real;
         Weight_zero : Real;
         Weight_Formula_W_T : Real;
         Visible : Bool;
         p_zero : Real;
         p_weight : Real;
         Zero_but : Bool;
         Weight_but : Bool;
         S : Real;
         Densyty : Real;
         Korect : Bool;
      END_STRUCT;
      "9_pol" : Struct
         Weight_db : Real;
         Weight_zero : Real;
         Weight_Formula_W_T : Real;
         Visible : Bool;
         p_zero : Real;
         p_weight : Real;
         Zero_but : Bool;
         Weight_but : Bool;
         S : Real;
         Densyty : Real;
         Korect : Bool;
      END_STRUCT;
      "10_pol" : Struct
         Weight_db : Real;
         Weight_zero : Real;
         Weight_Formula_W_T : Real;
         Visible : Bool;
         p_zero : Real;
         p_weight : Real;
         Zero_but : Bool;
         Weight_but : Bool;
         S : Real;
         Densyty : Real;
         Korect : Bool;
      END_STRUCT;
   END_STRUCT;


BEGIN
   Pol_p := 1.149812;
   Eror_pol_p := 16#0000_0000;
   S_pol := 6.819987;
   Weigt := 79.9358;
   Densyty := 1.35;
   "1_pol".Weight_db := 0.0;
   "1_pol".Weight_zero := 0.0;
   "1_pol".Weight_Formula_W_T := 81.81128;
   "1_pol".Visible := TRUE;
   "1_pol".p_zero := 0.0;
   "1_pol".p_weight := 0.0;
   "1_pol".Zero_but := FALSE;
   "1_pol".Weight_but := FALSE;
   "1_pol".S := 6.98;
   "1_pol".Densyty := 1.35;
   "1_pol".Korect := FALSE;
   "2_pol".Weight_db := 19.52373;
   "2_pol".Weight_zero := 0.0;
   "2_pol".Weight_Formula_W_T := 78.76387;
   "2_pol".Visible := FALSE;
   "2_pol".p_zero := 0.0;
   "2_pol".p_weight := 0.2850116;
   "2_pol".Zero_but := FALSE;
   "2_pol".Weight_but := FALSE;
   "2_pol".S := 6.72;
   "2_pol".Densyty := 1.35;
   "2_pol".Korect := FALSE;
   "3_pol".Weight_db := 0.0;
   "3_pol".Weight_zero := 0.0;
   "3_pol".Weight_Formula_W_T := 78.52945;
   "3_pol".Visible := FALSE;
   "3_pol".p_zero := 0.0;
   "3_pol".p_weight := 0.0;
   "3_pol".Zero_but := FALSE;
   "3_pol".Weight_but := FALSE;
   "3_pol".S := 6.7;
   "3_pol".Densyty := 1.35;
   "3_pol".Korect := FALSE;
   "4_pol".Weight_db := 73.68473;
   "4_pol".Weight_zero := 0.0;
   "4_pol".Weight_Formula_W_T := 78.76387;
   "4_pol".Visible := FALSE;
   "4_pol".p_zero := 0.0;
   "4_pol".p_weight := 1.075665;
   "4_pol".Zero_but := FALSE;
   "4_pol".Weight_but := FALSE;
   "4_pol".S := 6.72;
   "4_pol".Densyty := 1.35;
   "4_pol".Korect := FALSE;
   "5_pol".Weight_db := 24.61529;
   "5_pol".Weight_zero := 0.0;
   "5_pol".Weight_Formula_W_T := 77.55404;
   "5_pol".Visible := FALSE;
   "5_pol".p_zero := 0.0;
   "5_pol".p_weight := 0.364945;
   "5_pol".Zero_but := FALSE;
   "5_pol".Weight_but := FALSE;
   "5_pol".S := 6.61678;
   "5_pol".Densyty := 1.35;
   "5_pol".Korect := FALSE;
   "6_pol".Weight_db := 49.182;
   "6_pol".Weight_zero := 0.0;
   "6_pol".Weight_Formula_W_T := 78.64666;
   "6_pol".Visible := FALSE;
   "6_pol".p_zero := 0.0;
   "6_pol".p_weight := 0.7190394;
   "6_pol".Zero_but := FALSE;
   "6_pol".Weight_but := FALSE;
   "6_pol".S := 6.71;
   "6_pol".Densyty := 1.35;
   "6_pol".Korect := FALSE;
   "7_pol".Weight_db := 123.4003;
   "7_pol".Weight_zero := 0.0;
   "7_pol".Weight_Formula_W_T := 78.64666;
   "7_pol".Visible := FALSE;
   "7_pol".p_zero := 0.0;
   "7_pol".p_weight := 1.804109;
   "7_pol".Zero_but := FALSE;
   "7_pol".Weight_but := FALSE;
   "7_pol".S := 6.71;
   "7_pol".Densyty := 1.35;
   "7_pol".Korect := FALSE;
   "8_pol".Weight_db := -0.2724785;
   "8_pol".Weight_zero := 0.4211032;
   "8_pol".Weight_Formula_W_T := 78.74628;
   "8_pol".Visible := FALSE;
   "8_pol".p_zero := 0.006148727;
   "8_pol".p_weight := 0.002170139;
   "8_pol".Zero_but := FALSE;
   "8_pol".Weight_but := FALSE;
   "8_pol".S := 6.7185;
   "8_pol".Densyty := 1.35;
   "8_pol".Korect := FALSE;
   "9_pol".Weight_db := 126.8467;
   "9_pol".Weight_zero := 0.0;
   "9_pol".Weight_Formula_W_T := 78.97484;
   "9_pol".Visible := FALSE;
   "9_pol".p_zero := 0.0;
   "9_pol".p_weight := 1.846788;
   "9_pol".Zero_but := FALSE;
   "9_pol".Weight_but := FALSE;
   "9_pol".S := 6.738;
   "9_pol".Densyty := 1.35;
   "9_pol".Korect := FALSE;
   "10_pol".Weight_db := 27.88432;
   "10_pol".Weight_zero := 0.0;
   "10_pol".Weight_Formula_W_T := 77.55404;
   "10_pol".Visible := TRUE;
   "10_pol".p_zero := 0.0;
   "10_pol".p_weight := 0.4134114;
   "10_pol".Zero_but := FALSE;
   "10_pol".Weight_but := FALSE;
   "10_pol".S := 6.61678;
   "10_pol".Densyty := 1.35;
   "10_pol".Korect := FALSE;

END_DATA_BLOCK

DATA_BLOCK "iDB_Map_Siwarex_Core"
{ S7_Optimized_Access := 'FALSE' }
AUTHOR : S7C_Lib
FAMILY : Analog
VERSION : 1.4
"FB_Map_Siwarex_Core"

BEGIN

END_DATA_BLOCK

DATA_BLOCK "iFB_Map_Siwarex_Core"
{ S7_Optimized_Access := 'FALSE' }
AUTHOR : S7C_Lib
FAMILY : Analog
VERSION : 1.4
"FB_Map_Siwarex_Core"

BEGIN

END_DATA_BLOCK

DATA_BLOCK "MaxLevels"
{ S7_Optimized_Access := 'FALSE' }
VERSION : 0.1
   STRUCT 
      MaxLevel_Tank_1 : Real;
      MaxLevel_Tank_2 : Real;
      MaxLevel_Tank_3 : Real;
      MaxLevel_Tank_4 : Real;
      MaxLevel_Tank_5 : Real;
      MaxLevel_Tank_6 : Real;
      MaxLevel_Tank_7 : Real;
      MaxLevel_Tank_8 : Real;
      MaxLevel_Tank_9 : Real;
      MaxLevel_Tank_10 : Real;
      MaxLevel_Tank_11 : Real;
      MaxLevel_Tank_12 : Real;
      MaxLevel_Tank_13 : Real;
      MaxLevel_Tank_14 : Real;
   END_STRUCT;


BEGIN
   MaxLevel_Tank_1 := 15.0;
   MaxLevel_Tank_2 := 15.0;
   MaxLevel_Tank_3 := 15.0;
   MaxLevel_Tank_4 := 15.0;
   MaxLevel_Tank_5 := 15.0;
   MaxLevel_Tank_6 := 15.0;
   MaxLevel_Tank_7 := 15.0;
   MaxLevel_Tank_8 := 15.0;
   MaxLevel_Tank_9 := 15.0;
   MaxLevel_Tank_10 := 15.0;
   MaxLevel_Tank_11 := 13.0;
   MaxLevel_Tank_12 := 13.0;
   MaxLevel_Tank_13 := 13.0;
   MaxLevel_Tank_14 := 13.0;

END_DATA_BLOCK

DATA_BLOCK "DB_VECTOR_CS_1"
{ S7_Optimized_Access := 'FALSE' }
VERSION : 0.1
   STRUCT 
      lenghtdb : Int;
      POS_CMD601 : Int;
      POS_CMD602 : Int;
      POS_CMD603 : Int;
      POS_CMD604 : Int;
      POS_CMD605 : Int;
      POS_CMD606 : Int;
      POS_CMD607 : Int;
      POS_CMD608 : Int;
      POS_CMD609 : Int;
      POS_CMD610 : Int;
      DR3 : Struct
         number : Byte;
         lenght : Byte;
         adress : Int;
      END_STRUCT;
      DR4 : Struct
         number : Byte;
         lenght : Byte;
         adress : Int;
      END_STRUCT;
      DR9 : Struct
         number : Byte;
         lenght : Byte;
         adress : Int;
      END_STRUCT;
      DR15 : Struct
         number : Byte;
         lenght : Byte;
         adress : Int;
      END_STRUCT;
      DR26 : Struct
         number : Byte;
         lenght : Byte;
         adress : Int;
      END_STRUCT;
      DR30 : Struct
         number : Byte;
         lenght : Byte;
         adress : Int;
      END_STRUCT;
      DR0 : Struct
         number : Byte;
         lenght : Byte;
         adress : Int;
      END_STRUCT;
      LCMD605 : Byte;
      DR1CMD605 : Byte;
      DR2CMD605 : Byte;
      DR5CMD605 : Byte;
      DR6CMD605 : Byte;
      DR11CMD605 : Byte;
      DR12CMD605 : Byte;
      CMDCMD605 : Byte;
      LCMD610 : Byte;
      DR1CMD610 : Byte;
      DR2CMD610 : Byte;
      DR5CMD610 : Byte;
      DR6CMD610 : Byte;
      CMDCMD610 : Byte;
      lendbe : Int;
   END_STRUCT;


BEGIN
   lenghtdb := 66;
   POS_CMD601 := 0;
   POS_CMD602 := 0;
   POS_CMD603 := 0;
   POS_CMD604 := 0;
   POS_CMD605 := 50;
   POS_CMD606 := 0;
   POS_CMD607 := 0;
   POS_CMD608 := 0;
   POS_CMD609 := 0;
   POS_CMD610 := 58;
   DR3.number := 16#03;
   DR3.lenght := 16#38;
   DR3.adress := 50;
   DR4.number := 16#04;
   DR4.lenght := 16#0A;
   DR4.adress := 106;
   DR9.number := 16#09;
   DR9.lenght := 16#2C;
   DR9.adress := 116;
   DR15.number := 16#0F;
   DR15.lenght := 16#02;
   DR15.adress := 160;
   DR26.number := 16#1A;
   DR26.lenght := 16#0C;
   DR26.adress := 162;
   DR30.number := 16#1E;
   DR30.lenght := 16#2E;
   DR30.adress := 174;
   DR0.number := 16#00;
   DR0.lenght := 16#00;
   DR0.adress := 0;
   LCMD605 := 16#07;
   DR1CMD605 := 16#03;
   DR2CMD605 := 16#04;
   DR5CMD605 := 16#09;
   DR6CMD605 := 16#0F;
   DR11CMD605 := 16#1A;
   DR12CMD605 := 16#1E;
   CMDCMD605 := 16#00;
   LCMD610 := 16#05;
   DR1CMD610 := 16#03;
   DR2CMD610 := 16#04;
   DR5CMD610 := 16#0F;
   DR6CMD610 := 16#1A;
   CMDCMD610 := 16#00;
   lendbe := 66;

END_DATA_BLOCK

DATA_BLOCK "DB_VECTOR_CS_2"
{ S7_Optimized_Access := 'FALSE' }
VERSION : 0.1
   STRUCT 
      lenghtdb : Int;
      POS_CMD601 : Int;
      POS_CMD602 : Int;
      POS_CMD603 : Int;
      POS_CMD604 : Int;
      POS_CMD605 : Int;
      POS_CMD606 : Int;
      POS_CMD607 : Int;
      POS_CMD608 : Int;
      POS_CMD609 : Int;
      POS_CMD610 : Int;
      DR3 : Struct
         number : Byte;
         lenght : Byte;
         adress : Int;
      END_STRUCT;
      DR4 : Struct
         number : Byte;
         lenght : Byte;
         adress : Int;
      END_STRUCT;
      DR9 : Struct
         number : Byte;
         lenght : Byte;
         adress : Int;
      END_STRUCT;
      DR15 : Struct
         number : Byte;
         lenght : Byte;
         adress : Int;
      END_STRUCT;
      DR26 : Struct
         number : Byte;
         lenght : Byte;
         adress : Int;
      END_STRUCT;
      DR30 : Struct
         number : Byte;
         lenght : Byte;
         adress : Int;
      END_STRUCT;
      DR0 : Struct
         number : Byte;
         lenght : Byte;
         adress : Int;
      END_STRUCT;
      LCMD605 : Byte;
      DR1CMD605 : Byte;
      DR2CMD605 : Byte;
      DR5CMD605 : Byte;
      DR6CMD605 : Byte;
      DR11CMD605 : Byte;
      DR12CMD605 : Byte;
      CMDCMD605 : Byte;
      LCMD610 : Byte;
      DR1CMD610 : Byte;
      DR2CMD610 : Byte;
      DR5CMD610 : Byte;
      DR6CMD610 : Byte;
      CMDCMD610 : Byte;
      lendbe : Int;
   END_STRUCT;


BEGIN
   lenghtdb := 66;
   POS_CMD601 := 0;
   POS_CMD602 := 0;
   POS_CMD603 := 0;
   POS_CMD604 := 0;
   POS_CMD605 := 50;
   POS_CMD606 := 0;
   POS_CMD607 := 0;
   POS_CMD608 := 0;
   POS_CMD609 := 0;
   POS_CMD610 := 58;
   DR3.number := 16#03;
   DR3.lenght := 16#38;
   DR3.adress := 50;
   DR4.number := 16#04;
   DR4.lenght := 16#0A;
   DR4.adress := 106;
   DR9.number := 16#09;
   DR9.lenght := 16#2C;
   DR9.adress := 116;
   DR15.number := 16#0F;
   DR15.lenght := 16#02;
   DR15.adress := 160;
   DR26.number := 16#1A;
   DR26.lenght := 16#0C;
   DR26.adress := 162;
   DR30.number := 16#1E;
   DR30.lenght := 16#2E;
   DR30.adress := 174;
   DR0.number := 16#00;
   DR0.lenght := 16#00;
   DR0.adress := 0;
   LCMD605 := 16#07;
   DR1CMD605 := 16#03;
   DR2CMD605 := 16#04;
   DR5CMD605 := 16#09;
   DR6CMD605 := 16#0F;
   DR11CMD605 := 16#1A;
   DR12CMD605 := 16#1E;
   CMDCMD605 := 16#00;
   LCMD610 := 16#05;
   DR1CMD610 := 16#03;
   DR2CMD610 := 16#04;
   DR5CMD610 := 16#0F;
   DR6CMD610 := 16#1A;
   CMDCMD610 := 16#00;
   lendbe := 66;

END_DATA_BLOCK

DATA_BLOCK "FB_SICS_DR_T1"
{ S7_Optimized_Access := 'FALSE' }
AUTHOR : AD
FAMILY : SIWAREX
NAME : SICS_DR
VERSION : 2.0
"SICS_DR"

BEGIN
   ADDR := 260;
   DB_SCALE := 21;
   DB_VECTOR := 60;
   CMD_IN := 230;
   SEL_PROC_VAL := 16#00;
   EXT_TARA := 0;
   CMD_INPR := TRUE;
   CMD_FOK := FALSE;
   CMD_ERR := FALSE;
   CMD_ERR_C := 16#00;
   REF_COUNT := 16#4A;
   ACT_SEL_PROC_VAL := 16#00;
   PROC_VAL1 := 220;
   SC_STATUS := 16#00C0;
   ERR_MSG_C := 16#00;
   FB_ERR := FALSE;
   FB_ERR_C := 16#00;
   START_UP := FALSE;
   CMD_EN := TRUE;
   sb_CMD_EN_OLD := TRUE;
   sb_DI_OLD := FALSE;
   sb_BI_OLD := FALSE;
   sb_DIQ := FALSE;
   sb_BIQ := FALSE;
   sb_LB_OLD := FALSE;
   sb_AF_OLD := FALSE;
   sb_WRITE_DS := FALSE;
   sb_SFC_ERR := FALSE;
   si_CMD_IN_NEW := 0;
   si_CMD_IN_OLD := 230;
   si_ANZ_DS := 0;
   si_NEXT_ADR := 0;
   si_LB_CNT := 1;
   sy_CMD := 16#00;
   sy_DS_NO := 16#1E;
   sw_IN := 16#004A;
   sb_CMD_ERR_C := 16#00;
   si_ADR_DS := 42;
   si_TMP_SFC_ERR_CNT := 0;
   ss_APPL_ID := 'SIWAREX CS';
   sb_APPL_ID_ERR := FALSE;
   RDREC_1.REQ := TRUE;
   RDREC_1.ID := 16#0000_0104;
   RDREC_1.INDEX := 30;
   RDREC_1.MLEN := 46;
   RDREC_1.VALID := FALSE;
   RDREC_1.BUSY := TRUE;
   RDREC_1.ERROR := FALSE;
   RDREC_1.STATUS := 16#0070_0200;
   RDREC_1.LEN := 0;
   RDREC_1.RECORD := P#DB21.DBX174.0 BYTE 46;
   WRREC_1.REQ := FALSE;
   WRREC_1.ID := 16#0000_0000;
   WRREC_1.INDEX := 0;
   WRREC_1.LEN := 0;
   WRREC_1.DONE := FALSE;
   WRREC_1.BUSY := FALSE;
   WRREC_1.ERROR := FALSE;
   WRREC_1.STATUS := 16#0000_0000;
   WRREC_1.RECORD := NULL;
   MAX_CMD_OHNE_LS := 199;
   MAX_LESE_DS := 399;
   MAX_SCHREIBE_DS := 600;
   MAX_LESE_DS_VOR_CMD := 605;
   MAX_SCHREIBE_DS_VOR_CMD := 610;
   ADR_ANZ_ZYKLEN_LIFE_BIT := 2;
   ADR_RET_VAL_SFC58_59 := 4;
   ADR_TMP_SFC_ERR_CNT := 48;
   c_CMD_ERR_ANLAUF := 16#77;
   c_CMD_ERR_C_DR_CMD := 16#11;
   c_CMD_KETTE_ABGEB := 16#00;
   c_LB_CMD_ABBRUCH := 16#00;
   c_START_DR_DB_VECTOR := 18;

END_DATA_BLOCK

DATA_BLOCK "FB_SICS_DR_T2"
{ S7_Optimized_Access := 'FALSE' }
AUTHOR : AD
FAMILY : SIWAREX
NAME : SICS_DR
VERSION : 2.2
"SICS_DR"

BEGIN
   ADDR := 280;
   DB_SCALE := 62;
   DB_VECTOR := 63;
   CMD_IN := 230;
   SEL_PROC_VAL := 16#00;
   EXT_TARA := 0;
   CMD_INPR := TRUE;
   CMD_FOK := FALSE;
   CMD_ERR := FALSE;
   CMD_ERR_C := 16#00;
   REF_COUNT := 16#01;
   ACT_SEL_PROC_VAL := 16#00;
   PROC_VAL1 := -25;
   SC_STATUS := 16#02C0;
   ERR_MSG_C := 16#00;
   FB_ERR := FALSE;
   FB_ERR_C := 16#00;
   START_UP := FALSE;
   CMD_EN := TRUE;
   sb_CMD_EN_OLD := TRUE;
   sb_DI_OLD := FALSE;
   sb_BI_OLD := FALSE;
   sb_DIQ := FALSE;
   sb_BIQ := FALSE;
   sb_LB_OLD := TRUE;
   sb_AF_OLD := FALSE;
   sb_WRITE_DS := FALSE;
   sb_SFC_ERR := FALSE;
   si_CMD_IN_NEW := 0;
   si_CMD_IN_OLD := 230;
   si_ANZ_DS := 0;
   si_NEXT_ADR := 0;
   si_LB_CNT := 1;
   sy_CMD := 16#00;
   sy_DS_NO := 16#1E;
   sw_IN := 16#0401;
   sb_CMD_ERR_C := 16#00;
   si_ADR_DS := 42;
   si_TMP_SFC_ERR_CNT := 0;
   ss_APPL_ID := 'SIWAREX CS';
   sb_APPL_ID_ERR := FALSE;
   RDREC_1.REQ := TRUE;
   RDREC_1.ID := 16#0000_0118;
   RDREC_1.INDEX := 30;
   RDREC_1.MLEN := 46;
   RDREC_1.VALID := FALSE;
   RDREC_1.BUSY := TRUE;
   RDREC_1.ERROR := FALSE;
   RDREC_1.STATUS := 16#0070_0200;
   RDREC_1.LEN := 0;
   RDREC_1.RECORD := P#DB62.DBX174.0 BYTE 46;
   WRREC_1.REQ := FALSE;
   WRREC_1.ID := 16#0000_0000;
   WRREC_1.INDEX := 0;
   WRREC_1.LEN := 0;
   WRREC_1.DONE := FALSE;
   WRREC_1.BUSY := FALSE;
   WRREC_1.ERROR := FALSE;
   WRREC_1.STATUS := 16#0000_0000;
   WRREC_1.RECORD := NULL;
   MAX_CMD_OHNE_LS := 199;
   MAX_LESE_DS := 399;
   MAX_SCHREIBE_DS := 600;
   MAX_LESE_DS_VOR_CMD := 605;
   MAX_SCHREIBE_DS_VOR_CMD := 610;
   ADR_ANZ_ZYKLEN_LIFE_BIT := 2;
   ADR_RET_VAL_SFC58_59 := 4;
   ADR_TMP_SFC_ERR_CNT := 48;
   c_CMD_ERR_ANLAUF := 16#77;
   c_CMD_ERR_C_DR_CMD := 16#11;
   c_CMD_KETTE_ABGEB := 16#00;
   c_LB_CMD_ABBRUCH := 16#00;
   c_START_DR_DB_VECTOR := 18;

END_DATA_BLOCK

DATA_BLOCK "SICS_DR_DB"
{ S7_Optimized_Access := 'FALSE' }
AUTHOR : AD
FAMILY : SIWAREX
NAME : SICS_DR
VERSION : 2.2
"SICS_DR"

BEGIN
   ADDR := 0;
   DB_SCALE := 0;
   DB_VECTOR := 0;
   CMD_IN := 0;
   SEL_PROC_VAL := 16#00;
   EXT_TARA := 0;
   CMD_INPR := FALSE;
   CMD_FOK := FALSE;
   CMD_ERR := FALSE;
   CMD_ERR_C := 16#00;
   REF_COUNT := 16#00;
   ACT_SEL_PROC_VAL := 16#00;
   PROC_VAL1 := 0;
   SC_STATUS := 16#0000;
   ERR_MSG_C := 16#00;
   FB_ERR := FALSE;
   FB_ERR_C := 16#00;
   START_UP := FALSE;
   CMD_EN := FALSE;
   sb_CMD_EN_OLD := FALSE;
   sb_DI_OLD := FALSE;
   sb_BI_OLD := FALSE;
   sb_DIQ := FALSE;
   sb_BIQ := FALSE;
   sb_LB_OLD := FALSE;
   sb_AF_OLD := FALSE;
   sb_WRITE_DS := FALSE;
   sb_SFC_ERR := FALSE;
   si_CMD_IN_NEW := 0;
   si_CMD_IN_OLD := 0;
   si_ANZ_DS := 0;
   si_NEXT_ADR := 0;
   si_LB_CNT := 0;
   sy_CMD := 16#00;
   sy_DS_NO := 16#00;
   sw_IN := 16#0000;
   sb_CMD_ERR_C := 16#00;
   si_ADR_DS := 0;
   si_TMP_SFC_ERR_CNT := 0;
   ss_APPL_ID := 'SIWAREX CS';
   sb_APPL_ID_ERR := FALSE;
   RDREC_1.REQ := FALSE;
   RDREC_1.ID := 16#0000_0000;
   RDREC_1.INDEX := 0;
   RDREC_1.MLEN := 0;
   RDREC_1.VALID := FALSE;
   RDREC_1.BUSY := FALSE;
   RDREC_1.ERROR := FALSE;
   RDREC_1.STATUS := 16#0000_0000;
   RDREC_1.LEN := 0;
   RDREC_1.RECORD := NULL;
   WRREC_1.REQ := FALSE;
   WRREC_1.ID := 16#0000_0000;
   WRREC_1.INDEX := 0;
   WRREC_1.LEN := 0;
   WRREC_1.DONE := FALSE;
   WRREC_1.BUSY := FALSE;
   WRREC_1.ERROR := FALSE;
   WRREC_1.STATUS := 16#0000_0000;
   WRREC_1.RECORD := NULL;
   MAX_CMD_OHNE_LS := 0;
   MAX_LESE_DS := 0;
   MAX_SCHREIBE_DS := 0;
   MAX_LESE_DS_VOR_CMD := 0;
   MAX_SCHREIBE_DS_VOR_CMD := 0;
   ADR_ANZ_ZYKLEN_LIFE_BIT := 0;
   ADR_RET_VAL_SFC58_59 := 0;
   ADR_TMP_SFC_ERR_CNT := 0;
   c_CMD_ERR_ANLAUF := 16#00;
   c_CMD_ERR_C_DR_CMD := 16#00;
   c_CMD_KETTE_ABGEB := 16#00;
   c_LB_CMD_ABBRUCH := 16#00;
   c_START_DR_DB_VECTOR := 0;

END_DATA_BLOCK

DATA_BLOCK "iDB_Map_Siwarex_Core_1"
{ S7_Optimized_Access := 'FALSE' }
AUTHOR : S7C_Lib
FAMILY : Analog
VERSION : 1.4
"FB_Map_Siwarex_Core"

BEGIN

END_DATA_BLOCK

DATA_BLOCK "AI_Tank1_DB"
{ S7_Optimized_Access := 'FALSE' }
AUTHOR : SimenCom
VERSION : 1.0
"Analog_In_UDT"

BEGIN

END_DATA_BLOCK

DATA_BLOCK "CalcVolume_Tank1_DB"
{ S7_Optimized_Access := 'FALSE' }
VERSION : 0.1
"CalculationVolume"

BEGIN
   IW_Radius := 1.465;
   IW_ValueFromSensor := 17.53111;
   IW_K_for_Tonnag := 1.35;
   IW_K_for_Level := 1.35;
   QW_Volume := 87.51459;
   QW_Tonnag := 118.1447;
   QW_RealLevel := 12.986;
   sW_S := 6.739147;
   sW_Volume := 87.51459;
   sW_RealLevel := 12.986;

END_DATA_BLOCK

DATA_BLOCK "UDT_AI_Tank1"
{ S7_Optimized_Access := 'FALSE' }
VERSION : 0.1
"UDT_Analog_In"

BEGIN
   IW_HW_UpLevel := 27648;
   IW_HW_LowLevel := 0;
   IDW_UpLevel := 25.0;
   IDW_LowLevel := 0.0;
   IDW_HiHi := 4.0;
   IDW_Hi := 0.0;
   IDW_Lo := 0.0;
   IDW_Lolo := 0.0;
   IW_DelayON_HiHi := 0;
   IW_DelayON_Hi := 0;
   IW_DelayON_Lo := 0;
   IW_DelayON_LoLo := 0;
   IDW_Simulation_Value := 0.0;
   IW_Time_Filter := 0;
   IW_CTW[0] := FALSE;
   IW_CTW[1] := FALSE;
   IW_CTW[2] := FALSE;
   IW_CTW[3] := FALSE;
   IW_CTW[4] := FALSE;
   IW_CTW[5] := FALSE;
   IW_CTW[6] := FALSE;
   IW_CTW[7] := FALSE;
   IW_CTW[8] := FALSE;
   IW_CTW[9] := FALSE;
   IW_CTW[10] := FALSE;
   IW_CTW[11] := FALSE;
   IW_CTW[12] := FALSE;
   IW_CTW[13] := FALSE;
   IW_CTW[14] := FALSE;
   IW_CTW[15] := FALSE;
   IDW_K_Mult := 1.0;
   IDW_DeadZone := 0.0;
   IBt_Enable_ControlLevel[0] := FALSE;
   IBt_Enable_ControlLevel[1] := FALSE;
   IBt_Enable_ControlLevel[2] := FALSE;
   IBt_Enable_ControlLevel[3] := FALSE;
   IBt_Enable_ControlLevel[4] := FALSE;
   IBt_Enable_ControlLevel[5] := FALSE;
   IBt_Enable_ControlLevel[6] := FALSE;
   IBt_Enable_ControlLevel[7] := FALSE;
   IBt_Block_ControlLevel[0] := FALSE;
   IBt_Block_ControlLevel[1] := FALSE;
   IBt_Block_ControlLevel[2] := FALSE;
   IBt_Block_ControlLevel[3] := FALSE;
   IBt_Block_ControlLevel[4] := FALSE;
   IBt_Block_ControlLevel[5] := FALSE;
   IBt_Block_ControlLevel[6] := FALSE;
   IBt_Block_ControlLevel[7] := FALSE;
   QW_STW[0] := FALSE;
   QW_STW[1] := FALSE;
   QW_STW[2] := TRUE;
   QW_STW[3] := FALSE;
   QW_STW[4] := FALSE;
   QW_STW[5] := FALSE;
   QW_STW[6] := FALSE;
   QW_STW[7] := FALSE;
   QW_STW[8] := FALSE;
   QW_STW[9] := FALSE;
   QW_STW[10] := FALSE;
   QW_STW[11] := FALSE;
   QW_STW[12] := FALSE;
   QW_STW[13] := FALSE;
   QW_STW[14] := FALSE;
   QW_STW[15] := FALSE;
   QW_HWValue := 19388;
   QDW_ScalledValue := 17.53111;
   QDW_Message[0] := FALSE;
   QDW_Message[1] := FALSE;
   QDW_Message[2] := FALSE;
   QDW_Message[3] := FALSE;
   QDW_Message[4] := FALSE;
   QDW_Message[5] := FALSE;
   QDW_Message[6] := FALSE;
   QDW_Message[7] := FALSE;
   QDW_Message[8] := FALSE;
   QDW_Message[9] := FALSE;
   QDW_Message[10] := FALSE;
   QDW_Message[11] := FALSE;
   QDW_Message[12] := FALSE;
   QDW_Message[13] := FALSE;
   QDW_Message[14] := FALSE;
   QDW_Message[15] := FALSE;
   QDW_Message[16] := FALSE;

END_DATA_BLOCK

DATA_BLOCK "AI_Tank10_DB"
{ S7_Optimized_Access := 'FALSE' }
AUTHOR : SimenCom
VERSION : 1.0
"Analog_In_UDT"

BEGIN

END_DATA_BLOCK

DATA_BLOCK "CalcVolume_Tank10_DB"
{ S7_Optimized_Access := 'FALSE' }
VERSION : 0.1
"CalculationVolume"

BEGIN
   IW_Radius := 1.468;
   IW_ValueFromSensor := 18.56192;
   IW_K_for_Tonnag := 1.35;
   IW_K_for_Level := 1.35;
   QW_Volume := 93.04028;
   QW_Tonnag := 125.6044;
   QW_RealLevel := 13.74957;
   sW_S := 6.766776;
   sW_Volume := 93.04028;
   sW_RealLevel := 13.74957;

END_DATA_BLOCK

DATA_BLOCK "UDT_AI_Tank10"
{ S7_Optimized_Access := 'FALSE' }
VERSION : 0.1
"UDT_Analog_In"

BEGIN
   IW_HW_UpLevel := 27648;
   IW_HW_LowLevel := 0;
   IDW_UpLevel := 25.0;
   IDW_LowLevel := 0.0;
   IDW_HiHi := 18.5;
   IDW_Hi := 18.0;
   IDW_Lo := 0.0;
   IDW_Lolo := 0.0;
   IW_DelayON_HiHi := 1;
   IW_DelayON_Hi := 1;
   IW_DelayON_Lo := 0;
   IW_DelayON_LoLo := 0;
   IDW_Simulation_Value := 0.0;
   IW_Time_Filter := 0;
   IW_CTW[0] := FALSE;
   IW_CTW[1] := FALSE;
   IW_CTW[2] := FALSE;
   IW_CTW[3] := FALSE;
   IW_CTW[4] := FALSE;
   IW_CTW[5] := FALSE;
   IW_CTW[6] := FALSE;
   IW_CTW[7] := FALSE;
   IW_CTW[8] := FALSE;
   IW_CTW[9] := FALSE;
   IW_CTW[10] := FALSE;
   IW_CTW[11] := FALSE;
   IW_CTW[12] := FALSE;
   IW_CTW[13] := FALSE;
   IW_CTW[14] := FALSE;
   IW_CTW[15] := FALSE;
   IDW_K_Mult := 1.0;
   IDW_DeadZone := 0.0;
   IBt_Enable_ControlLevel[0] := TRUE;
   IBt_Enable_ControlLevel[1] := TRUE;
   IBt_Enable_ControlLevel[2] := FALSE;
   IBt_Enable_ControlLevel[3] := FALSE;
   IBt_Enable_ControlLevel[4] := FALSE;
   IBt_Enable_ControlLevel[5] := FALSE;
   IBt_Enable_ControlLevel[6] := FALSE;
   IBt_Enable_ControlLevel[7] := FALSE;
   IBt_Block_ControlLevel[0] := FALSE;
   IBt_Block_ControlLevel[1] := FALSE;
   IBt_Block_ControlLevel[2] := FALSE;
   IBt_Block_ControlLevel[3] := FALSE;
   IBt_Block_ControlLevel[4] := FALSE;
   IBt_Block_ControlLevel[5] := FALSE;
   IBt_Block_ControlLevel[6] := FALSE;
   IBt_Block_ControlLevel[7] := FALSE;
   QW_STW[0] := TRUE;
   QW_STW[1] := TRUE;
   QW_STW[2] := FALSE;
   QW_STW[3] := FALSE;
   QW_STW[4] := TRUE;
   QW_STW[5] := TRUE;
   QW_STW[6] := FALSE;
   QW_STW[7] := FALSE;
   QW_STW[8] := FALSE;
   QW_STW[9] := FALSE;
   QW_STW[10] := FALSE;
   QW_STW[11] := FALSE;
   QW_STW[12] := FALSE;
   QW_STW[13] := FALSE;
   QW_STW[14] := FALSE;
   QW_STW[15] := FALSE;
   QW_HWValue := 20524;
   QDW_ScalledValue := 18.5583;
   QDW_Message[0] := FALSE;
   QDW_Message[1] := TRUE;
   QDW_Message[2] := FALSE;
   QDW_Message[3] := FALSE;
   QDW_Message[4] := FALSE;
   QDW_Message[5] := FALSE;
   QDW_Message[6] := FALSE;
   QDW_Message[7] := FALSE;
   QDW_Message[8] := FALSE;
   QDW_Message[9] := FALSE;
   QDW_Message[10] := FALSE;
   QDW_Message[11] := FALSE;
   QDW_Message[12] := FALSE;
   QDW_Message[13] := FALSE;
   QDW_Message[14] := TRUE;
   QDW_Message[15] := FALSE;
   QDW_Message[16] := FALSE;

END_DATA_BLOCK

DATA_BLOCK "AI_Tank11_DB"
{ S7_Optimized_Access := 'FALSE' }
AUTHOR : SimenCom
VERSION : 1.0
"Analog_In_UDT"

BEGIN

END_DATA_BLOCK

DATA_BLOCK "CalcVolume_Tank11_DB"
{ S7_Optimized_Access := 'FALSE' }
VERSION : 0.1
"CalculationVolume"

BEGIN
   IW_Radius := 3.102;
   IW_ValueFromSensor := 6.546586;
   IW_K_for_Tonnag := 1.35;
   IW_K_for_Level := 1.35;
   QW_Volume := 146.5191;
   QW_Tonnag := 197.8008;
   QW_RealLevel := 4.849322;
   sW_S := 30.21435;
   sW_Volume := 146.5191;
   sW_RealLevel := 4.849322;

END_DATA_BLOCK

DATA_BLOCK "UDT_AI_Tank11"
{ S7_Optimized_Access := 'FALSE' }
VERSION : 0.1
"UDT_Analog_In"

BEGIN
   IW_HW_UpLevel := 27648;
   IW_HW_LowLevel := 0;
   IDW_UpLevel := 25.0;
   IDW_LowLevel := 0.0;
   IDW_HiHi := 17.5;
   IDW_Hi := 17.0;
   IDW_Lo := 0.0;
   IDW_Lolo := 0.0;
   IW_DelayON_HiHi := 1;
   IW_DelayON_Hi := 1;
   IW_DelayON_Lo := 0;
   IW_DelayON_LoLo := 0;
   IDW_Simulation_Value := 0.0;
   IW_Time_Filter := 0;
   IW_CTW[0] := FALSE;
   IW_CTW[1] := FALSE;
   IW_CTW[2] := FALSE;
   IW_CTW[3] := FALSE;
   IW_CTW[4] := FALSE;
   IW_CTW[5] := FALSE;
   IW_CTW[6] := FALSE;
   IW_CTW[7] := FALSE;
   IW_CTW[8] := FALSE;
   IW_CTW[9] := FALSE;
   IW_CTW[10] := FALSE;
   IW_CTW[11] := FALSE;
   IW_CTW[12] := FALSE;
   IW_CTW[13] := FALSE;
   IW_CTW[14] := FALSE;
   IW_CTW[15] := FALSE;
   IDW_K_Mult := 1.0;
   IDW_DeadZone := 0.0;
   IBt_Enable_ControlLevel[0] := TRUE;
   IBt_Enable_ControlLevel[1] := TRUE;
   IBt_Enable_ControlLevel[2] := FALSE;
   IBt_Enable_ControlLevel[3] := FALSE;
   IBt_Enable_ControlLevel[4] := FALSE;
   IBt_Enable_ControlLevel[5] := FALSE;
   IBt_Enable_ControlLevel[6] := FALSE;
   IBt_Enable_ControlLevel[7] := FALSE;
   IBt_Block_ControlLevel[0] := FALSE;
   IBt_Block_ControlLevel[1] := FALSE;
   IBt_Block_ControlLevel[2] := FALSE;
   IBt_Block_ControlLevel[3] := FALSE;
   IBt_Block_ControlLevel[4] := FALSE;
   IBt_Block_ControlLevel[5] := FALSE;
   IBt_Block_ControlLevel[6] := FALSE;
   IBt_Block_ControlLevel[7] := FALSE;
   QW_STW[0] := FALSE;
   QW_STW[1] := FALSE;
   QW_STW[2] := TRUE;
   QW_STW[3] := FALSE;
   QW_STW[4] := FALSE;
   QW_STW[5] := FALSE;
   QW_STW[6] := FALSE;
   QW_STW[7] := FALSE;
   QW_STW[8] := FALSE;
   QW_STW[9] := FALSE;
   QW_STW[10] := FALSE;
   QW_STW[11] := FALSE;
   QW_STW[12] := FALSE;
   QW_STW[13] := FALSE;
   QW_STW[14] := FALSE;
   QW_STW[15] := FALSE;
   QW_HWValue := 7240;
   QDW_ScalledValue := 6.546586;
   QDW_Message[0] := FALSE;
   QDW_Message[1] := FALSE;
   QDW_Message[2] := FALSE;
   QDW_Message[3] := FALSE;
   QDW_Message[4] := FALSE;
   QDW_Message[5] := FALSE;
   QDW_Message[6] := FALSE;
   QDW_Message[7] := FALSE;
   QDW_Message[8] := FALSE;
   QDW_Message[9] := FALSE;
   QDW_Message[10] := FALSE;
   QDW_Message[11] := FALSE;
   QDW_Message[12] := FALSE;
   QDW_Message[13] := FALSE;
   QDW_Message[14] := FALSE;
   QDW_Message[15] := FALSE;
   QDW_Message[16] := FALSE;

END_DATA_BLOCK

DATA_BLOCK "AI_Tank12_DB"
{ S7_Optimized_Access := 'FALSE' }
AUTHOR : SimenCom
VERSION : 1.0
"Analog_In_UDT"

BEGIN

END_DATA_BLOCK

DATA_BLOCK "CalcVolume_Tank12_DB"
{ S7_Optimized_Access := 'FALSE' }
VERSION : 0.1
"CalculationVolume"

BEGIN
   IW_Radius := 3.102;
   IW_ValueFromSensor := 15.90712;
   IW_K_for_Tonnag := 1.35;
   IW_K_for_Level := 1.35;
   QW_Volume := 356.0172;
   QW_Tonnag := 480.6232;
   QW_RealLevel := 11.78305;
   sW_S := 30.21435;
   sW_Volume := 356.0172;
   sW_RealLevel := 11.78305;

END_DATA_BLOCK

DATA_BLOCK "UDT_AI_Tank12"
{ S7_Optimized_Access := 'FALSE' }
VERSION : 0.1
"UDT_Analog_In"

BEGIN
   IW_HW_UpLevel := 27648;
   IW_HW_LowLevel := 0;
   IDW_UpLevel := 25.0;
   IDW_LowLevel := 0.0;
   IDW_HiHi := 17.5;
   IDW_Hi := 17.0;
   IDW_Lo := 0.0;
   IDW_Lolo := 0.0;
   IW_DelayON_HiHi := 1;
   IW_DelayON_Hi := 1;
   IW_DelayON_Lo := 0;
   IW_DelayON_LoLo := 0;
   IDW_Simulation_Value := 0.0;
   IW_Time_Filter := 0;
   IW_CTW[0] := FALSE;
   IW_CTW[1] := FALSE;
   IW_CTW[2] := FALSE;
   IW_CTW[3] := FALSE;
   IW_CTW[4] := FALSE;
   IW_CTW[5] := FALSE;
   IW_CTW[6] := FALSE;
   IW_CTW[7] := FALSE;
   IW_CTW[8] := FALSE;
   IW_CTW[9] := FALSE;
   IW_CTW[10] := FALSE;
   IW_CTW[11] := FALSE;
   IW_CTW[12] := FALSE;
   IW_CTW[13] := FALSE;
   IW_CTW[14] := FALSE;
   IW_CTW[15] := FALSE;
   IDW_K_Mult := 1.0;
   IDW_DeadZone := 0.0;
   IBt_Enable_ControlLevel[0] := TRUE;
   IBt_Enable_ControlLevel[1] := TRUE;
   IBt_Enable_ControlLevel[2] := FALSE;
   IBt_Enable_ControlLevel[3] := FALSE;
   IBt_Enable_ControlLevel[4] := FALSE;
   IBt_Enable_ControlLevel[5] := FALSE;
   IBt_Enable_ControlLevel[6] := FALSE;
   IBt_Enable_ControlLevel[7] := FALSE;
   IBt_Block_ControlLevel[0] := FALSE;
   IBt_Block_ControlLevel[1] := FALSE;
   IBt_Block_ControlLevel[2] := FALSE;
   IBt_Block_ControlLevel[3] := FALSE;
   IBt_Block_ControlLevel[4] := FALSE;
   IBt_Block_ControlLevel[5] := FALSE;
   IBt_Block_ControlLevel[6] := FALSE;
   IBt_Block_ControlLevel[7] := FALSE;
   QW_STW[0] := FALSE;
   QW_STW[1] := FALSE;
   QW_STW[2] := TRUE;
   QW_STW[3] := FALSE;
   QW_STW[4] := FALSE;
   QW_STW[5] := FALSE;
   QW_STW[6] := FALSE;
   QW_STW[7] := FALSE;
   QW_STW[8] := FALSE;
   QW_STW[9] := FALSE;
   QW_STW[10] := FALSE;
   QW_STW[11] := FALSE;
   QW_STW[12] := FALSE;
   QW_STW[13] := FALSE;
   QW_STW[14] := FALSE;
   QW_STW[15] := FALSE;
   QW_HWValue := 17592;
   QDW_ScalledValue := 15.90712;
   QDW_Message[0] := FALSE;
   QDW_Message[1] := FALSE;
   QDW_Message[2] := FALSE;
   QDW_Message[3] := FALSE;
   QDW_Message[4] := FALSE;
   QDW_Message[5] := FALSE;
   QDW_Message[6] := FALSE;
   QDW_Message[7] := FALSE;
   QDW_Message[8] := FALSE;
   QDW_Message[9] := FALSE;
   QDW_Message[10] := FALSE;
   QDW_Message[11] := FALSE;
   QDW_Message[12] := FALSE;
   QDW_Message[13] := FALSE;
   QDW_Message[14] := FALSE;
   QDW_Message[15] := FALSE;
   QDW_Message[16] := FALSE;

END_DATA_BLOCK

DATA_BLOCK "AI_Tank13_DB"
{ S7_Optimized_Access := 'FALSE' }
AUTHOR : SimenCom
VERSION : 1.0
"Analog_In_UDT"

BEGIN

END_DATA_BLOCK

DATA_BLOCK "CalcVolume_Tank13_DB"
{ S7_Optimized_Access := 'FALSE' }
VERSION : 0.1
"CalculationVolume"

BEGIN
   IW_Radius := 3.102;
   IW_ValueFromSensor := 5.385561;
   IW_K_for_Tonnag := 1.35;
   IW_K_for_Level := 1.35;
   QW_Volume := 120.5342;
   QW_Tonnag := 162.7212;
   QW_RealLevel := 3.989305;
   sW_S := 30.21435;
   sW_Volume := 120.5342;
   sW_RealLevel := 3.989305;

END_DATA_BLOCK

DATA_BLOCK "UDT_AI_Tank13"
{ S7_Optimized_Access := 'FALSE' }
VERSION : 0.1
"UDT_Analog_In"

BEGIN
   IW_HW_UpLevel := 27648;
   IW_HW_LowLevel := 0;
   IDW_UpLevel := 25.0;
   IDW_LowLevel := 0.0;
   IDW_HiHi := 17.5;
   IDW_Hi := 17.0;
   IDW_Lo := 0.0;
   IDW_Lolo := 0.0;
   IW_DelayON_HiHi := 1;
   IW_DelayON_Hi := 1;
   IW_DelayON_Lo := 0;
   IW_DelayON_LoLo := 0;
   IDW_Simulation_Value := 0.0;
   IW_Time_Filter := 0;
   IW_CTW[0] := FALSE;
   IW_CTW[1] := FALSE;
   IW_CTW[2] := FALSE;
   IW_CTW[3] := FALSE;
   IW_CTW[4] := FALSE;
   IW_CTW[5] := FALSE;
   IW_CTW[6] := FALSE;
   IW_CTW[7] := FALSE;
   IW_CTW[8] := FALSE;
   IW_CTW[9] := FALSE;
   IW_CTW[10] := FALSE;
   IW_CTW[11] := FALSE;
   IW_CTW[12] := FALSE;
   IW_CTW[13] := FALSE;
   IW_CTW[14] := FALSE;
   IW_CTW[15] := FALSE;
   IDW_K_Mult := 1.0;
   IDW_DeadZone := 0.0;
   IBt_Enable_ControlLevel[0] := TRUE;
   IBt_Enable_ControlLevel[1] := TRUE;
   IBt_Enable_ControlLevel[2] := FALSE;
   IBt_Enable_ControlLevel[3] := FALSE;
   IBt_Enable_ControlLevel[4] := FALSE;
   IBt_Enable_ControlLevel[5] := FALSE;
   IBt_Enable_ControlLevel[6] := FALSE;
   IBt_Enable_ControlLevel[7] := FALSE;
   IBt_Block_ControlLevel[0] := FALSE;
   IBt_Block_ControlLevel[1] := FALSE;
   IBt_Block_ControlLevel[2] := FALSE;
   IBt_Block_ControlLevel[3] := FALSE;
   IBt_Block_ControlLevel[4] := FALSE;
   IBt_Block_ControlLevel[5] := FALSE;
   IBt_Block_ControlLevel[6] := FALSE;
   IBt_Block_ControlLevel[7] := FALSE;
   QW_STW[0] := FALSE;
   QW_STW[1] := FALSE;
   QW_STW[2] := TRUE;
   QW_STW[3] := FALSE;
   QW_STW[4] := FALSE;
   QW_STW[5] := FALSE;
   QW_STW[6] := FALSE;
   QW_STW[7] := FALSE;
   QW_STW[8] := FALSE;
   QW_STW[9] := FALSE;
   QW_STW[10] := FALSE;
   QW_STW[11] := FALSE;
   QW_STW[12] := FALSE;
   QW_STW[13] := FALSE;
   QW_STW[14] := FALSE;
   QW_STW[15] := FALSE;
   QW_HWValue := 5952;
   QDW_ScalledValue := 5.381945;
   QDW_Message[0] := FALSE;
   QDW_Message[1] := FALSE;
   QDW_Message[2] := FALSE;
   QDW_Message[3] := FALSE;
   QDW_Message[4] := FALSE;
   QDW_Message[5] := FALSE;
   QDW_Message[6] := FALSE;
   QDW_Message[7] := FALSE;
   QDW_Message[8] := FALSE;
   QDW_Message[9] := FALSE;
   QDW_Message[10] := FALSE;
   QDW_Message[11] := FALSE;
   QDW_Message[12] := FALSE;
   QDW_Message[13] := FALSE;
   QDW_Message[14] := FALSE;
   QDW_Message[15] := FALSE;
   QDW_Message[16] := FALSE;

END_DATA_BLOCK

DATA_BLOCK "AI_Tank14_DB"
{ S7_Optimized_Access := 'FALSE' }
AUTHOR : SimenCom
VERSION : 1.0
"Analog_In_UDT"

BEGIN

END_DATA_BLOCK

DATA_BLOCK "CalcVolume_Tank14_DB"
{ S7_Optimized_Access := 'FALSE' }
VERSION : 0.1
"CalculationVolume"

BEGIN
   IW_Radius := 3.102;
   IW_ValueFromSensor := 17.18027;
   IW_K_for_Tonnag := 1.35;
   IW_K_for_Level := 1.35;
   QW_Volume := 384.5115;
   QW_Tonnag := 519.0905;
   QW_RealLevel := 12.72612;
   sW_S := 30.21435;
   sW_Volume := 384.5115;
   sW_RealLevel := 12.72612;

END_DATA_BLOCK

DATA_BLOCK "UDT_AI_Tank14"
{ S7_Optimized_Access := 'FALSE' }
VERSION : 0.1
"UDT_Analog_In"

BEGIN
   IW_HW_UpLevel := 27648;
   IW_HW_LowLevel := 0;
   IDW_UpLevel := 25.0;
   IDW_LowLevel := 0.0;
   IDW_HiHi := 17.5;
   IDW_Hi := 17.0;
   IDW_Lo := 0.0;
   IDW_Lolo := 0.0;
   IW_DelayON_HiHi := 1;
   IW_DelayON_Hi := 1;
   IW_DelayON_Lo := 0;
   IW_DelayON_LoLo := 0;
   IDW_Simulation_Value := 0.0;
   IW_Time_Filter := 0;
   IW_CTW[0] := FALSE;
   IW_CTW[1] := FALSE;
   IW_CTW[2] := FALSE;
   IW_CTW[3] := FALSE;
   IW_CTW[4] := FALSE;
   IW_CTW[5] := FALSE;
   IW_CTW[6] := FALSE;
   IW_CTW[7] := FALSE;
   IW_CTW[8] := FALSE;
   IW_CTW[9] := FALSE;
   IW_CTW[10] := FALSE;
   IW_CTW[11] := FALSE;
   IW_CTW[12] := FALSE;
   IW_CTW[13] := FALSE;
   IW_CTW[14] := FALSE;
   IW_CTW[15] := FALSE;
   IDW_K_Mult := 1.0;
   IDW_DeadZone := 0.0;
   IBt_Enable_ControlLevel[0] := TRUE;
   IBt_Enable_ControlLevel[1] := TRUE;
   IBt_Enable_ControlLevel[2] := FALSE;
   IBt_Enable_ControlLevel[3] := FALSE;
   IBt_Enable_ControlLevel[4] := FALSE;
   IBt_Enable_ControlLevel[5] := FALSE;
   IBt_Enable_ControlLevel[6] := FALSE;
   IBt_Enable_ControlLevel[7] := FALSE;
   IBt_Block_ControlLevel[0] := FALSE;
   IBt_Block_ControlLevel[1] := FALSE;
   IBt_Block_ControlLevel[2] := FALSE;
   IBt_Block_ControlLevel[3] := FALSE;
   IBt_Block_ControlLevel[4] := FALSE;
   IBt_Block_ControlLevel[5] := FALSE;
   IBt_Block_ControlLevel[6] := FALSE;
   IBt_Block_ControlLevel[7] := FALSE;
   QW_STW[0] := FALSE;
   QW_STW[1] := TRUE;
   QW_STW[2] := FALSE;
   QW_STW[3] := FALSE;
   QW_STW[4] := FALSE;
   QW_STW[5] := TRUE;
   QW_STW[6] := FALSE;
   QW_STW[7] := FALSE;
   QW_STW[8] := FALSE;
   QW_STW[9] := FALSE;
   QW_STW[10] := FALSE;
   QW_STW[11] := FALSE;
   QW_STW[12] := FALSE;
   QW_STW[13] := FALSE;
   QW_STW[14] := FALSE;
   QW_STW[15] := FALSE;
   QW_HWValue := 19000;
   QDW_ScalledValue := 17.18027;
   QDW_Message[0] := FALSE;
   QDW_Message[1] := FALSE;
   QDW_Message[2] := FALSE;
   QDW_Message[3] := FALSE;
   QDW_Message[4] := FALSE;
   QDW_Message[5] := FALSE;
   QDW_Message[6] := FALSE;
   QDW_Message[7] := FALSE;
   QDW_Message[8] := FALSE;
   QDW_Message[9] := FALSE;
   QDW_Message[10] := FALSE;
   QDW_Message[11] := FALSE;
   QDW_Message[12] := FALSE;
   QDW_Message[13] := FALSE;
   QDW_Message[14] := TRUE;
   QDW_Message[15] := FALSE;
   QDW_Message[16] := FALSE;

END_DATA_BLOCK

DATA_BLOCK "AI_Tank2_DB"
{ S7_Optimized_Access := 'FALSE' }
AUTHOR : SimenCom
VERSION : 1.0
"Analog_In_UDT"

BEGIN

END_DATA_BLOCK

DATA_BLOCK "CalcVolume_Tank2_DB"
{ S7_Optimized_Access := 'FALSE' }
VERSION : 0.1
"CalculationVolume"

BEGIN
   IW_Radius := 1.468;
   IW_ValueFromSensor := 18.41001;
   IW_K_for_Tonnag := 1.35;
   IW_K_for_Level := 1.35;
   QW_Volume := 92.27883;
   QW_Tonnag := 124.5764;
   QW_RealLevel := 13.63704;
   sW_S := 6.766776;
   sW_Volume := 92.27883;
   sW_RealLevel := 13.63704;

END_DATA_BLOCK

DATA_BLOCK "UDT_AI_Tank2"
{ S7_Optimized_Access := 'FALSE' }
VERSION : 0.1
"UDT_Analog_In"

BEGIN
   IW_HW_UpLevel := 27648;
   IW_HW_LowLevel := 0;
   IDW_UpLevel := 25.0;
   IDW_LowLevel := 0.0;
   IDW_HiHi := 18.5;
   IDW_Hi := 18.0;
   IDW_Lo := 0.0;
   IDW_Lolo := 0.0;
   IW_DelayON_HiHi := 1;
   IW_DelayON_Hi := 1;
   IW_DelayON_Lo := 0;
   IW_DelayON_LoLo := 0;
   IDW_Simulation_Value := 0.0;
   IW_Time_Filter := 0;
   IW_CTW[0] := FALSE;
   IW_CTW[1] := FALSE;
   IW_CTW[2] := FALSE;
   IW_CTW[3] := FALSE;
   IW_CTW[4] := FALSE;
   IW_CTW[5] := FALSE;
   IW_CTW[6] := FALSE;
   IW_CTW[7] := FALSE;
   IW_CTW[8] := FALSE;
   IW_CTW[9] := FALSE;
   IW_CTW[10] := FALSE;
   IW_CTW[11] := FALSE;
   IW_CTW[12] := FALSE;
   IW_CTW[13] := FALSE;
   IW_CTW[14] := FALSE;
   IW_CTW[15] := FALSE;
   IDW_K_Mult := 1.0;
   IDW_DeadZone := 0.0;
   IBt_Enable_ControlLevel[0] := FALSE;
   IBt_Enable_ControlLevel[1] := FALSE;
   IBt_Enable_ControlLevel[2] := FALSE;
   IBt_Enable_ControlLevel[3] := FALSE;
   IBt_Enable_ControlLevel[4] := FALSE;
   IBt_Enable_ControlLevel[5] := FALSE;
   IBt_Enable_ControlLevel[6] := FALSE;
   IBt_Enable_ControlLevel[7] := FALSE;
   IBt_Block_ControlLevel[0] := FALSE;
   IBt_Block_ControlLevel[1] := FALSE;
   IBt_Block_ControlLevel[2] := FALSE;
   IBt_Block_ControlLevel[3] := FALSE;
   IBt_Block_ControlLevel[4] := FALSE;
   IBt_Block_ControlLevel[5] := FALSE;
   IBt_Block_ControlLevel[6] := FALSE;
   IBt_Block_ControlLevel[7] := FALSE;
   QW_STW[0] := FALSE;
   QW_STW[1] := FALSE;
   QW_STW[2] := TRUE;
   QW_STW[3] := FALSE;
   QW_STW[4] := FALSE;
   QW_STW[5] := FALSE;
   QW_STW[6] := FALSE;
   QW_STW[7] := FALSE;
   QW_STW[8] := FALSE;
   QW_STW[9] := FALSE;
   QW_STW[10] := FALSE;
   QW_STW[11] := FALSE;
   QW_STW[12] := FALSE;
   QW_STW[13] := FALSE;
   QW_STW[14] := FALSE;
   QW_STW[15] := FALSE;
   QW_HWValue := 20356;
   QDW_ScalledValue := 18.40639;
   QDW_Message[0] := FALSE;
   QDW_Message[1] := FALSE;
   QDW_Message[2] := FALSE;
   QDW_Message[3] := FALSE;
   QDW_Message[4] := FALSE;
   QDW_Message[5] := FALSE;
   QDW_Message[6] := FALSE;
   QDW_Message[7] := FALSE;
   QDW_Message[8] := FALSE;
   QDW_Message[9] := FALSE;
   QDW_Message[10] := FALSE;
   QDW_Message[11] := FALSE;
   QDW_Message[12] := FALSE;
   QDW_Message[13] := FALSE;
   QDW_Message[14] := FALSE;
   QDW_Message[15] := FALSE;
   QDW_Message[16] := FALSE;

END_DATA_BLOCK

DATA_BLOCK "AI_Tank3_DB"
{ S7_Optimized_Access := 'FALSE' }
AUTHOR : SimenCom
VERSION : 1.0
"Analog_In_UDT"

BEGIN

END_DATA_BLOCK

DATA_BLOCK "CalcVolume_Tank3_DB"
{ S7_Optimized_Access := 'FALSE' }
VERSION : 0.1
"CalculationVolume"

BEGIN
   IW_Radius := 1.468;
   IW_ValueFromSensor := 9.675202;
   IW_K_for_Tonnag := 1.35;
   IW_K_for_Level := 1.35;
   QW_Volume := 48.49624;
   QW_Tonnag := 65.46992;
   QW_RealLevel := 7.166816;
   sW_S := 6.766776;
   sW_Volume := 48.49624;
   sW_RealLevel := 7.166816;

END_DATA_BLOCK

DATA_BLOCK "UDT_AI_Tank3"
{ S7_Optimized_Access := 'FALSE' }
VERSION : 0.1
"UDT_Analog_In"

BEGIN
   IW_HW_UpLevel := 27648;
   IW_HW_LowLevel := 0;
   IDW_UpLevel := 25.0;
   IDW_LowLevel := 0.0;
   IDW_HiHi := 18.5;
   IDW_Hi := 18.0;
   IDW_Lo := 0.0;
   IDW_Lolo := 4.0;
   IW_DelayON_HiHi := 1;
   IW_DelayON_Hi := 1;
   IW_DelayON_Lo := 0;
   IW_DelayON_LoLo := 0;
   IDW_Simulation_Value := 0.0;
   IW_Time_Filter := 0;
   IW_CTW[0] := FALSE;
   IW_CTW[1] := FALSE;
   IW_CTW[2] := FALSE;
   IW_CTW[3] := FALSE;
   IW_CTW[4] := FALSE;
   IW_CTW[5] := FALSE;
   IW_CTW[6] := FALSE;
   IW_CTW[7] := FALSE;
   IW_CTW[8] := FALSE;
   IW_CTW[9] := FALSE;
   IW_CTW[10] := FALSE;
   IW_CTW[11] := FALSE;
   IW_CTW[12] := FALSE;
   IW_CTW[13] := FALSE;
   IW_CTW[14] := FALSE;
   IW_CTW[15] := FALSE;
   IDW_K_Mult := 1.0;
   IDW_DeadZone := 0.0;
   IBt_Enable_ControlLevel[0] := TRUE;
   IBt_Enable_ControlLevel[1] := TRUE;
   IBt_Enable_ControlLevel[2] := FALSE;
   IBt_Enable_ControlLevel[3] := FALSE;
   IBt_Enable_ControlLevel[4] := FALSE;
   IBt_Enable_ControlLevel[5] := FALSE;
   IBt_Enable_ControlLevel[6] := FALSE;
   IBt_Enable_ControlLevel[7] := FALSE;
   IBt_Block_ControlLevel[0] := FALSE;
   IBt_Block_ControlLevel[1] := FALSE;
   IBt_Block_ControlLevel[2] := FALSE;
   IBt_Block_ControlLevel[3] := FALSE;
   IBt_Block_ControlLevel[4] := FALSE;
   IBt_Block_ControlLevel[5] := FALSE;
   IBt_Block_ControlLevel[6] := FALSE;
   IBt_Block_ControlLevel[7] := FALSE;
   QW_STW[0] := FALSE;
   QW_STW[1] := FALSE;
   QW_STW[2] := TRUE;
   QW_STW[3] := FALSE;
   QW_STW[4] := FALSE;
   QW_STW[5] := FALSE;
   QW_STW[6] := FALSE;
   QW_STW[7] := FALSE;
   QW_STW[8] := FALSE;
   QW_STW[9] := FALSE;
   QW_STW[10] := FALSE;
   QW_STW[11] := FALSE;
   QW_STW[12] := FALSE;
   QW_STW[13] := FALSE;
   QW_STW[14] := FALSE;
   QW_STW[15] := FALSE;
   QW_HWValue := 10704;
   QDW_ScalledValue := 9.67882;
   QDW_Message[0] := FALSE;
   QDW_Message[1] := FALSE;
   QDW_Message[2] := FALSE;
   QDW_Message[3] := FALSE;
   QDW_Message[4] := FALSE;
   QDW_Message[5] := FALSE;
   QDW_Message[6] := FALSE;
   QDW_Message[7] := FALSE;
   QDW_Message[8] := FALSE;
   QDW_Message[9] := FALSE;
   QDW_Message[10] := FALSE;
   QDW_Message[11] := FALSE;
   QDW_Message[12] := FALSE;
   QDW_Message[13] := FALSE;
   QDW_Message[14] := FALSE;
   QDW_Message[15] := FALSE;
   QDW_Message[16] := FALSE;

END_DATA_BLOCK

DATA_BLOCK "AI_Tank4_DB"
{ S7_Optimized_Access := 'FALSE' }
AUTHOR : SimenCom
VERSION : 1.0
"Analog_In_UDT"

BEGIN

END_DATA_BLOCK

DATA_BLOCK "CalcVolume_Tank4_DB"
{ S7_Optimized_Access := 'FALSE' }
VERSION : 0.1
"CalculationVolume"

BEGIN
   IW_Radius := 1.468;
   IW_ValueFromSensor := 13.19083;
   IW_K_for_Tonnag := 1.35;
   IW_K_for_Level := 1.35;
   QW_Volume := 66.11805;
   QW_Tonnag := 89.25937;
   QW_RealLevel := 9.770983;
   sW_S := 6.766776;
   sW_Volume := 66.11805;
   sW_RealLevel := 9.770983;

END_DATA_BLOCK

DATA_BLOCK "UDT_AI_Tank4"
{ S7_Optimized_Access := 'FALSE' }
VERSION : 0.1
"UDT_Analog_In"

BEGIN
   IW_HW_UpLevel := 27648;
   IW_HW_LowLevel := 0;
   IDW_UpLevel := 25.0;
   IDW_LowLevel := 0.0;
   IDW_HiHi := 18.5;
   IDW_Hi := 18.0;
   IDW_Lo := 0.0;
   IDW_Lolo := 0.0;
   IW_DelayON_HiHi := 1;
   IW_DelayON_Hi := 1;
   IW_DelayON_Lo := 0;
   IW_DelayON_LoLo := 0;
   IDW_Simulation_Value := 0.0;
   IW_Time_Filter := 0;
   IW_CTW[0] := FALSE;
   IW_CTW[1] := FALSE;
   IW_CTW[2] := FALSE;
   IW_CTW[3] := FALSE;
   IW_CTW[4] := FALSE;
   IW_CTW[5] := FALSE;
   IW_CTW[6] := FALSE;
   IW_CTW[7] := FALSE;
   IW_CTW[8] := FALSE;
   IW_CTW[9] := FALSE;
   IW_CTW[10] := FALSE;
   IW_CTW[11] := FALSE;
   IW_CTW[12] := FALSE;
   IW_CTW[13] := FALSE;
   IW_CTW[14] := FALSE;
   IW_CTW[15] := FALSE;
   IDW_K_Mult := 1.0;
   IDW_DeadZone := 0.0;
   IBt_Enable_ControlLevel[0] := TRUE;
   IBt_Enable_ControlLevel[1] := TRUE;
   IBt_Enable_ControlLevel[2] := FALSE;
   IBt_Enable_ControlLevel[3] := FALSE;
   IBt_Enable_ControlLevel[4] := FALSE;
   IBt_Enable_ControlLevel[5] := FALSE;
   IBt_Enable_ControlLevel[6] := FALSE;
   IBt_Enable_ControlLevel[7] := FALSE;
   IBt_Block_ControlLevel[0] := FALSE;
   IBt_Block_ControlLevel[1] := FALSE;
   IBt_Block_ControlLevel[2] := FALSE;
   IBt_Block_ControlLevel[3] := FALSE;
   IBt_Block_ControlLevel[4] := FALSE;
   IBt_Block_ControlLevel[5] := FALSE;
   IBt_Block_ControlLevel[6] := FALSE;
   IBt_Block_ControlLevel[7] := FALSE;
   QW_STW[0] := FALSE;
   QW_STW[1] := FALSE;
   QW_STW[2] := TRUE;
   QW_STW[3] := FALSE;
   QW_STW[4] := FALSE;
   QW_STW[5] := FALSE;
   QW_STW[6] := FALSE;
   QW_STW[7] := FALSE;
   QW_STW[8] := FALSE;
   QW_STW[9] := FALSE;
   QW_STW[10] := FALSE;
   QW_STW[11] := FALSE;
   QW_STW[12] := FALSE;
   QW_STW[13] := FALSE;
   QW_STW[14] := FALSE;
   QW_STW[15] := FALSE;
   QW_HWValue := 14588;
   QDW_ScalledValue := 13.19083;
   QDW_Message[0] := FALSE;
   QDW_Message[1] := FALSE;
   QDW_Message[2] := FALSE;
   QDW_Message[3] := FALSE;
   QDW_Message[4] := FALSE;
   QDW_Message[5] := FALSE;
   QDW_Message[6] := FALSE;
   QDW_Message[7] := FALSE;
   QDW_Message[8] := FALSE;
   QDW_Message[9] := FALSE;
   QDW_Message[10] := FALSE;
   QDW_Message[11] := FALSE;
   QDW_Message[12] := FALSE;
   QDW_Message[13] := FALSE;
   QDW_Message[14] := FALSE;
   QDW_Message[15] := FALSE;
   QDW_Message[16] := FALSE;

END_DATA_BLOCK

DATA_BLOCK "AI_Tank5_DB"
{ S7_Optimized_Access := 'FALSE' }
AUTHOR : SimenCom
VERSION : 1.0
"Analog_In_UDT"

BEGIN

END_DATA_BLOCK

DATA_BLOCK "CalcVolume_Tank5_DB"
{ S7_Optimized_Access := 'FALSE' }
VERSION : 0.1
"CalculationVolume"

BEGIN
   IW_Radius := 1.468;
   IW_ValueFromSensor := 18.26172;
   IW_K_for_Tonnag := 1.35;
   IW_K_for_Level := 1.35;
   QW_Volume := 91.53552;
   QW_Tonnag := 123.573;
   QW_RealLevel := 13.5272;
   sW_S := 6.766776;
   sW_Volume := 91.53552;
   sW_RealLevel := 13.5272;

END_DATA_BLOCK

DATA_BLOCK "UDT_AI_Tank5"
{ S7_Optimized_Access := 'FALSE' }
VERSION : 0.1
"UDT_Analog_In"

BEGIN
   IW_HW_UpLevel := 27648;
   IW_HW_LowLevel := 0;
   IDW_UpLevel := 25.0;
   IDW_LowLevel := 0.0;
   IDW_HiHi := 18.5;
   IDW_Hi := 18.0;
   IDW_Lo := 0.0;
   IDW_Lolo := 0.0;
   IW_DelayON_HiHi := 1;
   IW_DelayON_Hi := 1;
   IW_DelayON_Lo := 0;
   IW_DelayON_LoLo := 0;
   IDW_Simulation_Value := 0.0;
   IW_Time_Filter := 0;
   IW_CTW[0] := FALSE;
   IW_CTW[1] := FALSE;
   IW_CTW[2] := FALSE;
   IW_CTW[3] := FALSE;
   IW_CTW[4] := FALSE;
   IW_CTW[5] := FALSE;
   IW_CTW[6] := FALSE;
   IW_CTW[7] := FALSE;
   IW_CTW[8] := FALSE;
   IW_CTW[9] := FALSE;
   IW_CTW[10] := FALSE;
   IW_CTW[11] := FALSE;
   IW_CTW[12] := FALSE;
   IW_CTW[13] := FALSE;
   IW_CTW[14] := FALSE;
   IW_CTW[15] := FALSE;
   IDW_K_Mult := 1.0;
   IDW_DeadZone := 0.0;
   IBt_Enable_ControlLevel[0] := TRUE;
   IBt_Enable_ControlLevel[1] := TRUE;
   IBt_Enable_ControlLevel[2] := FALSE;
   IBt_Enable_ControlLevel[3] := FALSE;
   IBt_Enable_ControlLevel[4] := FALSE;
   IBt_Enable_ControlLevel[5] := FALSE;
   IBt_Enable_ControlLevel[6] := FALSE;
   IBt_Enable_ControlLevel[7] := FALSE;
   IBt_Block_ControlLevel[0] := FALSE;
   IBt_Block_ControlLevel[1] := FALSE;
   IBt_Block_ControlLevel[2] := FALSE;
   IBt_Block_ControlLevel[3] := FALSE;
   IBt_Block_ControlLevel[4] := FALSE;
   IBt_Block_ControlLevel[5] := FALSE;
   IBt_Block_ControlLevel[6] := FALSE;
   IBt_Block_ControlLevel[7] := FALSE;
   QW_STW[0] := FALSE;
   QW_STW[1] := TRUE;
   QW_STW[2] := FALSE;
   QW_STW[3] := FALSE;
   QW_STW[4] := FALSE;
   QW_STW[5] := TRUE;
   QW_STW[6] := FALSE;
   QW_STW[7] := FALSE;
   QW_STW[8] := FALSE;
   QW_STW[9] := FALSE;
   QW_STW[10] := FALSE;
   QW_STW[11] := FALSE;
   QW_STW[12] := FALSE;
   QW_STW[13] := FALSE;
   QW_STW[14] := FALSE;
   QW_STW[15] := FALSE;
   QW_HWValue := 20196;
   QDW_ScalledValue := 18.26172;
   QDW_Message[0] := FALSE;
   QDW_Message[1] := FALSE;
   QDW_Message[2] := FALSE;
   QDW_Message[3] := FALSE;
   QDW_Message[4] := FALSE;
   QDW_Message[5] := FALSE;
   QDW_Message[6] := FALSE;
   QDW_Message[7] := FALSE;
   QDW_Message[8] := FALSE;
   QDW_Message[9] := FALSE;
   QDW_Message[10] := FALSE;
   QDW_Message[11] := FALSE;
   QDW_Message[12] := FALSE;
   QDW_Message[13] := FALSE;
   QDW_Message[14] := TRUE;
   QDW_Message[15] := FALSE;
   QDW_Message[16] := FALSE;

END_DATA_BLOCK

DATA_BLOCK "AI_Tank6_DB"
{ S7_Optimized_Access := 'FALSE' }
AUTHOR : SimenCom
VERSION : 1.0
"Analog_In_UDT"

BEGIN

END_DATA_BLOCK

DATA_BLOCK "CalcVolume_Tank6_DB"
{ S7_Optimized_Access := 'FALSE' }
VERSION : 0.1
"CalculationVolume"

BEGIN
   IW_Radius := 1.468;
   IW_ValueFromSensor := 18.24364;
   IW_K_for_Tonnag := 1.35;
   IW_K_for_Level := 1.35;
   QW_Volume := 91.44489;
   QW_Tonnag := 123.4506;
   QW_RealLevel := 13.5138;
   sW_S := 6.766776;
   sW_Volume := 91.44489;
   sW_RealLevel := 13.5138;

END_DATA_BLOCK

DATA_BLOCK "UDT_AI_Tank6"
{ S7_Optimized_Access := 'FALSE' }
VERSION : 0.1
"UDT_Analog_In"

BEGIN
   IW_HW_UpLevel := 27648;
   IW_HW_LowLevel := 0;
   IDW_UpLevel := 25.0;
   IDW_LowLevel := 0.0;
   IDW_HiHi := 18.5;
   IDW_Hi := 18.0;
   IDW_Lo := 0.0;
   IDW_Lolo := 0.0;
   IW_DelayON_HiHi := 1;
   IW_DelayON_Hi := 1;
   IW_DelayON_Lo := 0;
   IW_DelayON_LoLo := 0;
   IDW_Simulation_Value := 0.0;
   IW_Time_Filter := 0;
   IW_CTW[0] := FALSE;
   IW_CTW[1] := FALSE;
   IW_CTW[2] := FALSE;
   IW_CTW[3] := FALSE;
   IW_CTW[4] := FALSE;
   IW_CTW[5] := FALSE;
   IW_CTW[6] := FALSE;
   IW_CTW[7] := FALSE;
   IW_CTW[8] := FALSE;
   IW_CTW[9] := FALSE;
   IW_CTW[10] := FALSE;
   IW_CTW[11] := FALSE;
   IW_CTW[12] := FALSE;
   IW_CTW[13] := FALSE;
   IW_CTW[14] := FALSE;
   IW_CTW[15] := FALSE;
   IDW_K_Mult := 1.0;
   IDW_DeadZone := 0.0;
   IBt_Enable_ControlLevel[0] := TRUE;
   IBt_Enable_ControlLevel[1] := TRUE;
   IBt_Enable_ControlLevel[2] := FALSE;
   IBt_Enable_ControlLevel[3] := FALSE;
   IBt_Enable_ControlLevel[4] := FALSE;
   IBt_Enable_ControlLevel[5] := FALSE;
   IBt_Enable_ControlLevel[6] := FALSE;
   IBt_Enable_ControlLevel[7] := FALSE;
   IBt_Block_ControlLevel[0] := FALSE;
   IBt_Block_ControlLevel[1] := FALSE;
   IBt_Block_ControlLevel[2] := FALSE;
   IBt_Block_ControlLevel[3] := FALSE;
   IBt_Block_ControlLevel[4] := FALSE;
   IBt_Block_ControlLevel[5] := FALSE;
   IBt_Block_ControlLevel[6] := FALSE;
   IBt_Block_ControlLevel[7] := FALSE;
   QW_STW[0] := FALSE;
   QW_STW[1] := TRUE;
   QW_STW[2] := FALSE;
   QW_STW[3] := FALSE;
   QW_STW[4] := FALSE;
   QW_STW[5] := TRUE;
   QW_STW[6] := FALSE;
   QW_STW[7] := FALSE;
   QW_STW[8] := FALSE;
   QW_STW[9] := FALSE;
   QW_STW[10] := FALSE;
   QW_STW[11] := FALSE;
   QW_STW[12] := FALSE;
   QW_STW[13] := FALSE;
   QW_STW[14] := FALSE;
   QW_STW[15] := FALSE;
   QW_HWValue := 20172;
   QDW_ScalledValue := 18.24002;
   QDW_Message[0] := FALSE;
   QDW_Message[1] := FALSE;
   QDW_Message[2] := FALSE;
   QDW_Message[3] := FALSE;
   QDW_Message[4] := FALSE;
   QDW_Message[5] := FALSE;
   QDW_Message[6] := FALSE;
   QDW_Message[7] := FALSE;
   QDW_Message[8] := FALSE;
   QDW_Message[9] := FALSE;
   QDW_Message[10] := FALSE;
   QDW_Message[11] := FALSE;
   QDW_Message[12] := FALSE;
   QDW_Message[13] := FALSE;
   QDW_Message[14] := TRUE;
   QDW_Message[15] := FALSE;
   QDW_Message[16] := FALSE;

END_DATA_BLOCK

DATA_BLOCK "AI_Tank7_DB"
{ S7_Optimized_Access := 'FALSE' }
AUTHOR : SimenCom
VERSION : 1.0
"Analog_In_UDT"

BEGIN

END_DATA_BLOCK

DATA_BLOCK "CalcVolume_Tank7_DB"
{ S7_Optimized_Access := 'FALSE' }
VERSION : 0.1
"CalculationVolume"

BEGIN
   IW_Radius := 1.468;
   IW_ValueFromSensor := 13.7406;
   IW_K_for_Tonnag := 1.35;
   IW_K_for_Level := 1.35;
   QW_Volume := 68.87373;
   QW_Tonnag := 92.97953;
   QW_RealLevel := 10.17822;
   sW_S := 6.766776;
   sW_Volume := 68.87373;
   sW_RealLevel := 10.17822;

END_DATA_BLOCK

DATA_BLOCK "UDT_AI_Tank7"
{ S7_Optimized_Access := 'FALSE' }
VERSION : 0.1
"UDT_Analog_In"

BEGIN
   IW_HW_UpLevel := 27648;
   IW_HW_LowLevel := 0;
   IDW_UpLevel := 25.0;
   IDW_LowLevel := 0.0;
   IDW_HiHi := 18.5;
   IDW_Hi := 18.0;
   IDW_Lo := 0.0;
   IDW_Lolo := 0.0;
   IW_DelayON_HiHi := 1;
   IW_DelayON_Hi := 1;
   IW_DelayON_Lo := 0;
   IW_DelayON_LoLo := 0;
   IDW_Simulation_Value := 0.0;
   IW_Time_Filter := 0;
   IW_CTW[0] := FALSE;
   IW_CTW[1] := FALSE;
   IW_CTW[2] := FALSE;
   IW_CTW[3] := FALSE;
   IW_CTW[4] := FALSE;
   IW_CTW[5] := FALSE;
   IW_CTW[6] := FALSE;
   IW_CTW[7] := FALSE;
   IW_CTW[8] := FALSE;
   IW_CTW[9] := FALSE;
   IW_CTW[10] := FALSE;
   IW_CTW[11] := FALSE;
   IW_CTW[12] := FALSE;
   IW_CTW[13] := FALSE;
   IW_CTW[14] := FALSE;
   IW_CTW[15] := FALSE;
   IDW_K_Mult := 1.0;
   IDW_DeadZone := 0.0;
   IBt_Enable_ControlLevel[0] := TRUE;
   IBt_Enable_ControlLevel[1] := TRUE;
   IBt_Enable_ControlLevel[2] := FALSE;
   IBt_Enable_ControlLevel[3] := FALSE;
   IBt_Enable_ControlLevel[4] := FALSE;
   IBt_Enable_ControlLevel[5] := FALSE;
   IBt_Enable_ControlLevel[6] := FALSE;
   IBt_Enable_ControlLevel[7] := FALSE;
   IBt_Block_ControlLevel[0] := FALSE;
   IBt_Block_ControlLevel[1] := FALSE;
   IBt_Block_ControlLevel[2] := FALSE;
   IBt_Block_ControlLevel[3] := FALSE;
   IBt_Block_ControlLevel[4] := FALSE;
   IBt_Block_ControlLevel[5] := FALSE;
   IBt_Block_ControlLevel[6] := FALSE;
   IBt_Block_ControlLevel[7] := FALSE;
   QW_STW[0] := FALSE;
   QW_STW[1] := FALSE;
   QW_STW[2] := TRUE;
   QW_STW[3] := FALSE;
   QW_STW[4] := FALSE;
   QW_STW[5] := FALSE;
   QW_STW[6] := FALSE;
   QW_STW[7] := FALSE;
   QW_STW[8] := FALSE;
   QW_STW[9] := FALSE;
   QW_STW[10] := FALSE;
   QW_STW[11] := FALSE;
   QW_STW[12] := FALSE;
   QW_STW[13] := FALSE;
   QW_STW[14] := FALSE;
   QW_STW[15] := FALSE;
   QW_HWValue := 15200;
   QDW_ScalledValue := 13.74421;
   QDW_Message[0] := FALSE;
   QDW_Message[1] := FALSE;
   QDW_Message[2] := FALSE;
   QDW_Message[3] := FALSE;
   QDW_Message[4] := FALSE;
   QDW_Message[5] := FALSE;
   QDW_Message[6] := FALSE;
   QDW_Message[7] := FALSE;
   QDW_Message[8] := FALSE;
   QDW_Message[9] := FALSE;
   QDW_Message[10] := FALSE;
   QDW_Message[11] := FALSE;
   QDW_Message[12] := FALSE;
   QDW_Message[13] := FALSE;
   QDW_Message[14] := FALSE;
   QDW_Message[15] := FALSE;
   QDW_Message[16] := FALSE;

END_DATA_BLOCK

DATA_BLOCK "AI_Tank8_DB"
{ S7_Optimized_Access := 'FALSE' }
AUTHOR : SimenCom
VERSION : 1.0
"Analog_In_UDT"

BEGIN

END_DATA_BLOCK

DATA_BLOCK "CalcVolume_Tank8_DB"
{ S7_Optimized_Access := 'FALSE' }
VERSION : 0.1
"CalculationVolume"

BEGIN
   IW_Radius := 1.468;
   IW_ValueFromSensor := 18.48597;
   IW_K_for_Tonnag := 1.35;
   IW_K_for_Level := 1.35;
   QW_Volume := 92.65955;
   QW_Tonnag := 125.0904;
   QW_RealLevel := 13.69331;
   sW_S := 6.766776;
   sW_Volume := 92.65955;
   sW_RealLevel := 13.69331;

END_DATA_BLOCK

DATA_BLOCK "UDT_AI_Tank8"
{ S7_Optimized_Access := 'FALSE' }
VERSION : 0.1
"UDT_Analog_In"

BEGIN
   IW_HW_UpLevel := 27648;
   IW_HW_LowLevel := 0;
   IDW_UpLevel := 25.0;
   IDW_LowLevel := 0.0;
   IDW_HiHi := 18.5;
   IDW_Hi := 18.0;
   IDW_Lo := 0.0;
   IDW_Lolo := 0.0;
   IW_DelayON_HiHi := 1;
   IW_DelayON_Hi := 1;
   IW_DelayON_Lo := 0;
   IW_DelayON_LoLo := 0;
   IDW_Simulation_Value := 0.0;
   IW_Time_Filter := 0;
   IW_CTW[0] := FALSE;
   IW_CTW[1] := FALSE;
   IW_CTW[2] := FALSE;
   IW_CTW[3] := FALSE;
   IW_CTW[4] := FALSE;
   IW_CTW[5] := FALSE;
   IW_CTW[6] := FALSE;
   IW_CTW[7] := FALSE;
   IW_CTW[8] := FALSE;
   IW_CTW[9] := FALSE;
   IW_CTW[10] := FALSE;
   IW_CTW[11] := FALSE;
   IW_CTW[12] := FALSE;
   IW_CTW[13] := FALSE;
   IW_CTW[14] := FALSE;
   IW_CTW[15] := FALSE;
   IDW_K_Mult := 1.0;
   IDW_DeadZone := 0.0;
   IBt_Enable_ControlLevel[0] := TRUE;
   IBt_Enable_ControlLevel[1] := TRUE;
   IBt_Enable_ControlLevel[2] := FALSE;
   IBt_Enable_ControlLevel[3] := FALSE;
   IBt_Enable_ControlLevel[4] := FALSE;
   IBt_Enable_ControlLevel[5] := FALSE;
   IBt_Enable_ControlLevel[6] := FALSE;
   IBt_Enable_ControlLevel[7] := FALSE;
   IBt_Block_ControlLevel[0] := FALSE;
   IBt_Block_ControlLevel[1] := FALSE;
   IBt_Block_ControlLevel[2] := FALSE;
   IBt_Block_ControlLevel[3] := FALSE;
   IBt_Block_ControlLevel[4] := FALSE;
   IBt_Block_ControlLevel[5] := FALSE;
   IBt_Block_ControlLevel[6] := FALSE;
   IBt_Block_ControlLevel[7] := FALSE;
   QW_STW[0] := FALSE;
   QW_STW[1] := TRUE;
   QW_STW[2] := FALSE;
   QW_STW[3] := FALSE;
   QW_STW[4] := FALSE;
   QW_STW[5] := TRUE;
   QW_STW[6] := FALSE;
   QW_STW[7] := FALSE;
   QW_STW[8] := FALSE;
   QW_STW[9] := FALSE;
   QW_STW[10] := FALSE;
   QW_STW[11] := FALSE;
   QW_STW[12] := FALSE;
   QW_STW[13] := FALSE;
   QW_STW[14] := FALSE;
   QW_STW[15] := FALSE;
   QW_HWValue := 20444;
   QDW_ScalledValue := 18.48597;
   QDW_Message[0] := FALSE;
   QDW_Message[1] := FALSE;
   QDW_Message[2] := FALSE;
   QDW_Message[3] := FALSE;
   QDW_Message[4] := FALSE;
   QDW_Message[5] := FALSE;
   QDW_Message[6] := FALSE;
   QDW_Message[7] := FALSE;
   QDW_Message[8] := FALSE;
   QDW_Message[9] := FALSE;
   QDW_Message[10] := FALSE;
   QDW_Message[11] := FALSE;
   QDW_Message[12] := FALSE;
   QDW_Message[13] := FALSE;
   QDW_Message[14] := TRUE;
   QDW_Message[15] := FALSE;
   QDW_Message[16] := FALSE;

END_DATA_BLOCK

DATA_BLOCK "AI_Tank9_DB"
{ S7_Optimized_Access := 'FALSE' }
AUTHOR : SimenCom
VERSION : 1.0
"Analog_In_UDT"

BEGIN

END_DATA_BLOCK

DATA_BLOCK "CalcVolume_Tank9_DB"
{ S7_Optimized_Access := 'FALSE' }
VERSION : 0.1
"CalculationVolume"

BEGIN
   IW_Radius := 1.468;
   IW_ValueFromSensor := 18.20747;
   IW_K_for_Tonnag := 1.35;
   IW_K_for_Level := 1.35;
   QW_Volume := 91.26359;
   QW_Tonnag := 123.2058;
   QW_RealLevel := 13.48701;
   sW_S := 6.766776;
   sW_Volume := 91.26359;
   sW_RealLevel := 13.48701;

END_DATA_BLOCK

DATA_BLOCK "UDT_AI_Tank9"
{ S7_Optimized_Access := 'FALSE' }
VERSION : 0.1
"UDT_Analog_In"

BEGIN
   IW_HW_UpLevel := 27648;
   IW_HW_LowLevel := 0;
   IDW_UpLevel := 25.0;
   IDW_LowLevel := 0.0;
   IDW_HiHi := 18.5;
   IDW_Hi := 18.0;
   IDW_Lo := 0.0;
   IDW_Lolo := 0.0;
   IW_DelayON_HiHi := 1;
   IW_DelayON_Hi := 1;
   IW_DelayON_Lo := 0;
   IW_DelayON_LoLo := 0;
   IDW_Simulation_Value := 0.0;
   IW_Time_Filter := 0;
   IW_CTW[0] := FALSE;
   IW_CTW[1] := FALSE;
   IW_CTW[2] := FALSE;
   IW_CTW[3] := FALSE;
   IW_CTW[4] := FALSE;
   IW_CTW[5] := FALSE;
   IW_CTW[6] := FALSE;
   IW_CTW[7] := FALSE;
   IW_CTW[8] := FALSE;
   IW_CTW[9] := FALSE;
   IW_CTW[10] := FALSE;
   IW_CTW[11] := FALSE;
   IW_CTW[12] := FALSE;
   IW_CTW[13] := FALSE;
   IW_CTW[14] := FALSE;
   IW_CTW[15] := FALSE;
   IDW_K_Mult := 1.0;
   IDW_DeadZone := 0.0;
   IBt_Enable_ControlLevel[0] := TRUE;
   IBt_Enable_ControlLevel[1] := TRUE;
   IBt_Enable_ControlLevel[2] := FALSE;
   IBt_Enable_ControlLevel[3] := FALSE;
   IBt_Enable_ControlLevel[4] := FALSE;
   IBt_Enable_ControlLevel[5] := FALSE;
   IBt_Enable_ControlLevel[6] := FALSE;
   IBt_Enable_ControlLevel[7] := FALSE;
   IBt_Block_ControlLevel[0] := FALSE;
   IBt_Block_ControlLevel[1] := FALSE;
   IBt_Block_ControlLevel[2] := FALSE;
   IBt_Block_ControlLevel[3] := FALSE;
   IBt_Block_ControlLevel[4] := FALSE;
   IBt_Block_ControlLevel[5] := FALSE;
   IBt_Block_ControlLevel[6] := FALSE;
   IBt_Block_ControlLevel[7] := FALSE;
   QW_STW[0] := FALSE;
   QW_STW[1] := TRUE;
   QW_STW[2] := FALSE;
   QW_STW[3] := FALSE;
   QW_STW[4] := FALSE;
   QW_STW[5] := TRUE;
   QW_STW[6] := FALSE;
   QW_STW[7] := FALSE;
   QW_STW[8] := FALSE;
   QW_STW[9] := FALSE;
   QW_STW[10] := FALSE;
   QW_STW[11] := FALSE;
   QW_STW[12] := FALSE;
   QW_STW[13] := FALSE;
   QW_STW[14] := FALSE;
   QW_STW[15] := FALSE;
   QW_HWValue := 20136;
   QDW_ScalledValue := 18.20747;
   QDW_Message[0] := FALSE;
   QDW_Message[1] := FALSE;
   QDW_Message[2] := FALSE;
   QDW_Message[3] := FALSE;
   QDW_Message[4] := FALSE;
   QDW_Message[5] := FALSE;
   QDW_Message[6] := FALSE;
   QDW_Message[7] := FALSE;
   QDW_Message[8] := FALSE;
   QDW_Message[9] := FALSE;
   QDW_Message[10] := FALSE;
   QDW_Message[11] := FALSE;
   QDW_Message[12] := FALSE;
   QDW_Message[13] := FALSE;
   QDW_Message[14] := TRUE;
   QDW_Message[15] := FALSE;
   QDW_Message[16] := FALSE;

END_DATA_BLOCK

ORGANIZATION_BLOCK "Main"   // OB1, FBD, ProgramCycle
TITLE = "Main Program Sweep (Cycle)"
   VAR_TEMP
      OB1_EV_CLASS : Byte;   // Bits 0-3 = 1 (Coming event), Bits 4-7 = 1 (Event class 1)
      OB1_SCAN_1 : Byte;   // 1 (Cold restart scan 1 of OB 1), 3 (Scan 2-n of OB 1)
      OB1_PRIORITY : Byte;   // Priority of OB Execution
      OB1_OB_NUMBR : Byte;   // 1 (Organization block 1, OB1)
      OB1_RESERVED_1 : Byte;   // Reserved for system
      OB1_RESERVED_2 : Byte;   // Reserved for system
      OB1_PREV_CYCLE : Int;   // Cycle time of previous OB1 scan (milliseconds)
      OB1_MIN_CYCLE : Int;   // Minimum cycle time of OB1 (milliseconds)
      OB1_MAX_CYCLE : Int;   // Maximum cycle time of OB1 (milliseconds)
      OB1_DATE_TIME : Date_And_Time;   // Date and time OB1 started
   END_VAR
   VAR_TEMP   // added for the SCL form of the ladder/FBD networks
      _w1 : Bool;
   END_VAR
BEGIN

REGION Network 1
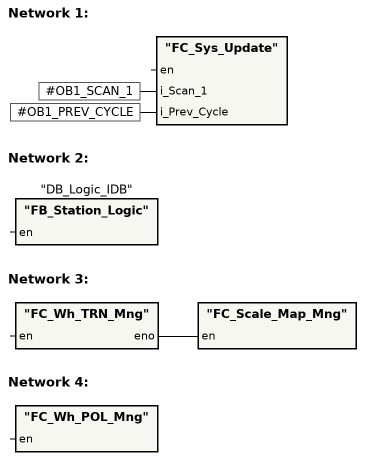
   "FC_Sys_Update"(i_Scan_1 := #OB1_SCAN_1, i_Prev_Cycle := #OB1_PREV_CYCLE);
END_REGION

REGION Network 2
   "DB_Logic_IDB"();   // "FB_Station_Logic"
END_REGION

REGION Network 3
   "FC_Wh_TRN_Mng"(ENO => #_w1);
   IF #_w1 THEN "FC_Scale_Map_Mng"(); END_IF;
END_REGION

REGION Network 4
   "FC_Wh_POL_Mng"();
END_REGION
END_ORGANIZATION_BLOCK

FUNCTION "FC_Sys_Update" : Void
{ S7_Optimized_Access := 'FALSE' }
VERSION : 0.1
// 3. SYSTEM FUNCTIONS
   VAR_INPUT 
      i_Scan_1 : Byte;
      i_Prev_Cycle : Int;
   END_VAR

   VAR_TEMP 
      tmp_dint : DInt;
   END_VAR


BEGIN
	"DB_Global".Sys.FirstScan := (#i_Scan_1 <> B#16#03);
	
	"DB_Global".Sys.CycleTime_ms_INT := #i_Prev_Cycle;
	IF #i_Prev_Cycle <= 0 THEN
	    #tmp_dint := 1;
	ELSE
	    #tmp_dint := INT_TO_DINT(#i_Prev_Cycle);
	END_IF;
	"DB_Global".Sys.CycleTime_ms_REAL := DINT_TO_REAL(#tmp_dint);
	
END_FUNCTION

FUNCTION_BLOCK "FB_Station_Logic"
{ S7_Optimized_Access := 'FALSE' }
VERSION : 0.1
// 6. WRAPPER FB (The only block with actual memory for instances)
   VAR 
      fb_Saw : "FB_Sim_SawTooth_UpDown";
      fb_Dist : "FB_RawDistort";
      AI_1 : "FB_AI";
      AI_2 : "FB_AI";
      Alarm_1 : "FB_AnalogAlarm";
      Alarm_2 : "FB_AnalogAlarm";
   END_VAR

   VAR_TEMP 
      tmp_raw_gen : Int;
   END_VAR


BEGIN
	
	#fb_Saw(Enable := "DB_Test_IO".Sim_Enable_Saw,
	        Speed := "DB_Test_IO".Sim_Saw_Speed,
	        Current_Val := "DB_Test_IO".Raw_Start,
	        Out_Raw => #tmp_raw_gen,
	        Limit_Low := "DB_Test_IO".Raw_Min,
	        Limit_High := "DB_Test_IO".Raw_Max);
	#fb_Dist(Enable := "DB_Test_IO".Sim_Enable_Noise,
	         RawIn := #tmp_raw_gen,
	         Dt_ms := "getCycleTime"(),
	         NoiseAmpRaw := "DB_Test_IO".Sim_Noise_Amp,
	         Noise_Hz := "DB_Test_IO".Sim_Noise_Hz,
	         RawOut => "DB_Test_IO".Raw_Final);
	
	#AI_1(i_iRawSignal := "DB_Test_IO".Raw_Final,
	      io_stConfig := "DB_Test_IO".Config[1],
	      io_stOut := "DB_Test_IO".Out[1]);
	#Alarm_1(
	         i_rValue := "DB_Test_IO".Out[1].Value_Filtered,
	         i_boReset := "DB_Test_IO".Reset_Alarms,
	         // Умная блокировка: глушим сирену, если отпал датчик, КЗ или кривые настройки
	         i_boInhibit := "DB_Test_IO".Out[1].Status.WireBreak OR
	                         "DB_Test_IO".Out[1].Status.Overflow OR
	                         "DB_Test_IO".Out[1].Status.ConfigError,
	         io_stConfig := "DB_Test_IO".Alarm_Cfg[1],
	         io_stOut := "DB_Test_IO".Alarm_Out[1]
	);
	
